// TIA Portal V17 export
// export: Created 2025-03-05T08:01:26.5756457Z, ExportSetting WithDefaults, DisplayName Totally Integrated Automation Portal, DisplayVersion V17 Update 8, DisplayName TIA Portal Openness, DisplayVersion V17 Update 8, DisplayName TIA Portal Version Control Interface, DisplayVersion V17, DisplayName SINAMICS Startdrive Advanced, DisplayVersion V17 SP2, DisplayName SINAMICS Startdrive G110M, G120, G120C, G120D, G120P, G115D, DisplayVersion V17 SP2, DisplayName SINAMICS Startdrive G130, G150, S120, S150, SINAMICS MV, S210, DisplayVersion V17 SP2, DisplayName STEP 7 Professional, DisplayVersion V17 Update 8, DisplayName SINUMERIK ONE STEP 7 Toolbox, DisplayVersion V17 Update 12, DisplayName SINUMERIK 840D sl STEP 7 Toolbox, DisplayVersion V17 Update 12, DisplayName STEP 7 Safety, DisplayVersion V17 Update 6, DisplayName WinCC Advanced, DisplayVersion V17 Update 8
FUNCTION "FC16015_METHOD_CALLS_U02_STA3_COAXIAL" : Void   // FC16015, LAD
{ S7_Optimized_Access := 'TRUE' }
VERSION : 0.1
// stored: AutoNumber false, IsIECCheckEnabled false, SetENOAutomatically false, UDAEnableTagReadback false
   VAR_TEMP
      AUX_WSTRING_PART_ID_STA3 : WString;
      AUX_WCHARS : Array[0..63] of WChar;
      index : Int;
      ALARM_AUX : Bool;
      TEMP_PULSE : Bool;
   END_VAR
   VAR_TEMP   // added for the SCL form of the ladder/FBD networks
      _w1 : Bool;
   END_VAR
BEGIN

REGION Network 1 (SCL): TRANSFORM TO WCHARS
   FOR #index := 0 TO 63 DO
       #AUX_WCHARS[#index] := CHAR_TO_WCHAR("DB8000_PART_STATUS".UNIT_02.STATION_3.PART_A.PART_ID[#index]);
   END_FOR;
END_REGION

REGION Network 2: TRANSFORM TO WSTRING
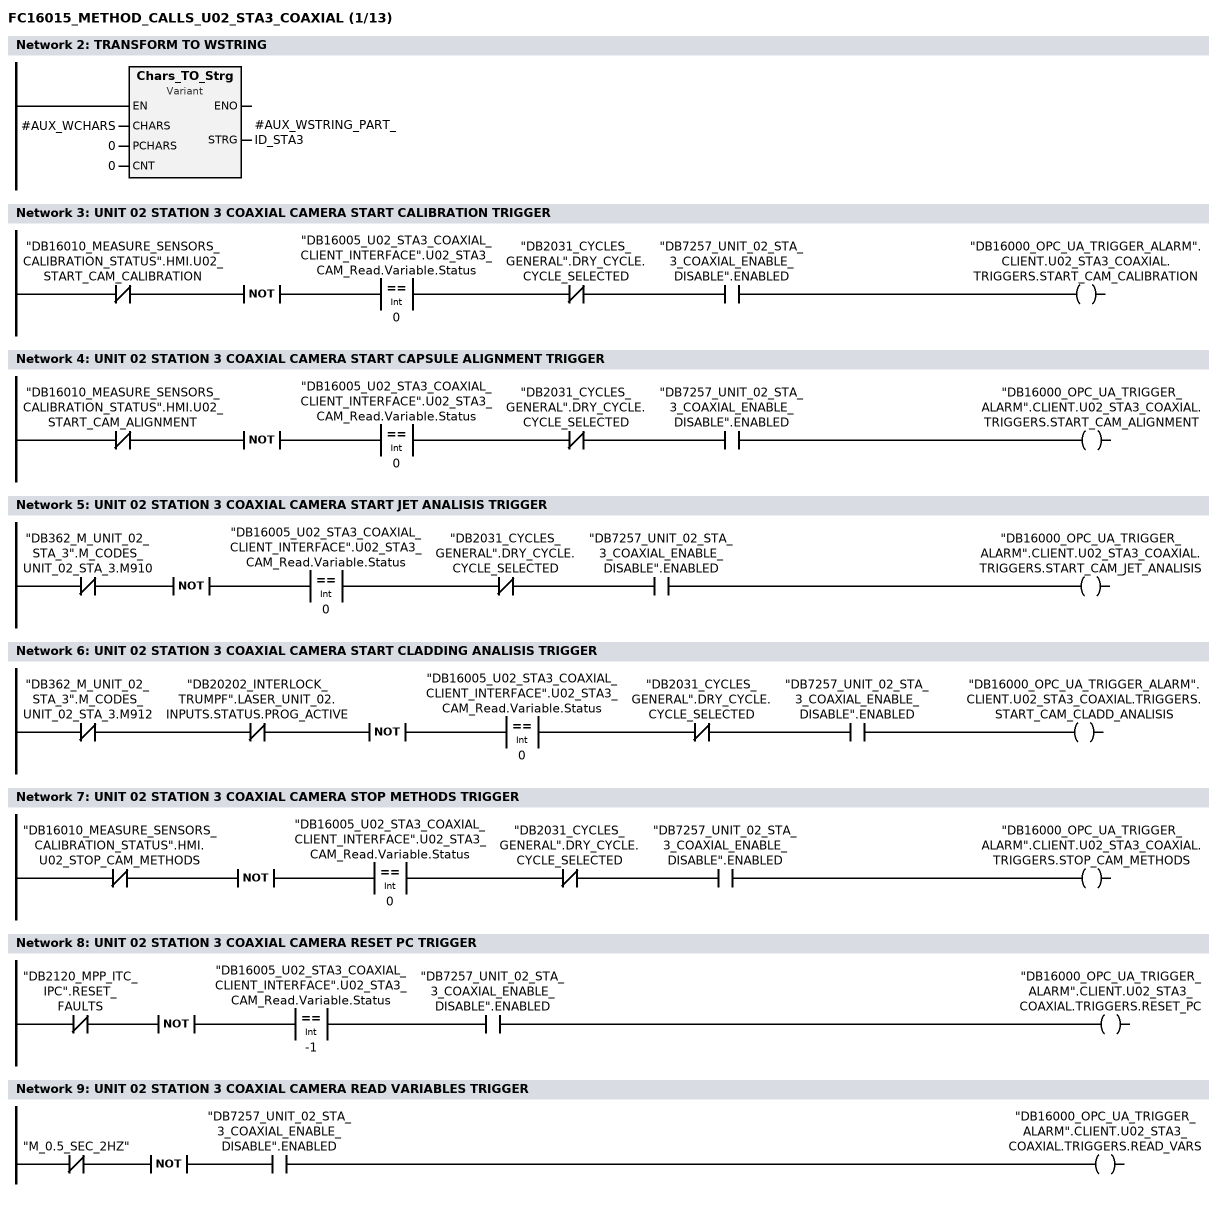
   RUNG wire#powerrail
      { S7_Templates := "[ptr_type := Variant, str_type := WString]" } Chars_TO_Strg(Chars := #AUX_WCHARS, pChars := 0, Cnt := 0, Strg => #AUX_WSTRING_PART_ID_STA3)
   END_RUNG
   // the same network as SCL:
   Chars_TO_Strg(Chars := #AUX_WCHARS, pChars := 0, Cnt := 0, Strg => #AUX_WSTRING_PART_ID_STA3);
END_REGION

REGION Network 3: UNIT 02 STATION 3 COAXIAL CAMERA START CALIBRATION TRIGGER
   RUNG wire#powerrail
      I_Contact( "DB16010_MEASURE_SENSORS_CALIBRATION_STATUS".HMI.U02_START_CAM_CALIBRATION )
      Not()
      { S7_Templates := "SrcType := Int" } EQ_Contact(in1 := "DB16005_U02_STA3_COAXIAL_CLIENT_INTERFACE".U02_STA3_CAM_Read.Variable.Status, in2 := 0)
      I_Contact( "DB2031_CYCLES_GENERAL".DRY_CYCLE.CYCLE_SELECTED )
      Contact( "DB7257_UNIT_02_STA_3_COAXIAL_ENABLE_DISABLE".ENABLED )
      Coil( "DB16000_OPC_UA_TRIGGER_ALARM".CLIENT.U02_STA3_COAXIAL.TRIGGERS.START_CAM_CALIBRATION )
   END_RUNG
   // the same network as SCL:
   "DB16000_OPC_UA_TRIGGER_ALARM".CLIENT.U02_STA3_COAXIAL.TRIGGERS.START_CAM_CALIBRATION := NOT (NOT "DB16010_MEASURE_SENSORS_CALIBRATION_STATUS".HMI.U02_START_CAM_CALIBRATION) AND ("DB16005_U02_STA3_COAXIAL_CLIENT_INTERFACE".U02_STA3_CAM_Read.Variable.Status = 0) AND NOT "DB2031_CYCLES_GENERAL".DRY_CYCLE.CYCLE_SELECTED AND "DB7257_UNIT_02_STA_3_COAXIAL_ENABLE_DISABLE".ENABLED;
END_REGION

REGION Network 4: UNIT 02 STATION 3 COAXIAL CAMERA START CAPSULE ALIGNMENT TRIGGER
   RUNG wire#powerrail
      I_Contact( "DB16010_MEASURE_SENSORS_CALIBRATION_STATUS".HMI.U02_START_CAM_ALIGNMENT )
      Not()
      { S7_Templates := "SrcType := Int" } EQ_Contact(in1 := "DB16005_U02_STA3_COAXIAL_CLIENT_INTERFACE".U02_STA3_CAM_Read.Variable.Status, in2 := 0)
      I_Contact( "DB2031_CYCLES_GENERAL".DRY_CYCLE.CYCLE_SELECTED )
      Contact( "DB7257_UNIT_02_STA_3_COAXIAL_ENABLE_DISABLE".ENABLED )
      Coil( "DB16000_OPC_UA_TRIGGER_ALARM".CLIENT.U02_STA3_COAXIAL.TRIGGERS.START_CAM_ALIGNMENT )
   END_RUNG
   // the same network as SCL:
   "DB16000_OPC_UA_TRIGGER_ALARM".CLIENT.U02_STA3_COAXIAL.TRIGGERS.START_CAM_ALIGNMENT := NOT (NOT "DB16010_MEASURE_SENSORS_CALIBRATION_STATUS".HMI.U02_START_CAM_ALIGNMENT) AND ("DB16005_U02_STA3_COAXIAL_CLIENT_INTERFACE".U02_STA3_CAM_Read.Variable.Status = 0) AND NOT "DB2031_CYCLES_GENERAL".DRY_CYCLE.CYCLE_SELECTED AND "DB7257_UNIT_02_STA_3_COAXIAL_ENABLE_DISABLE".ENABLED;
END_REGION

REGION Network 5: UNIT 02 STATION 3 COAXIAL CAMERA START JET ANALISIS TRIGGER
   RUNG wire#powerrail
      I_Contact( "DB362_M_UNIT_02_STA_3".M_CODES_UNIT_02_STA_3.M910 )
      Not()
      { S7_Templates := "SrcType := Int" } EQ_Contact(in1 := "DB16005_U02_STA3_COAXIAL_CLIENT_INTERFACE".U02_STA3_CAM_Read.Variable.Status, in2 := 0)
      I_Contact( "DB2031_CYCLES_GENERAL".DRY_CYCLE.CYCLE_SELECTED )
      Contact( "DB7257_UNIT_02_STA_3_COAXIAL_ENABLE_DISABLE".ENABLED )
      Coil( "DB16000_OPC_UA_TRIGGER_ALARM".CLIENT.U02_STA3_COAXIAL.TRIGGERS.START_CAM_JET_ANALISIS )
   END_RUNG
   // the same network as SCL:
   "DB16000_OPC_UA_TRIGGER_ALARM".CLIENT.U02_STA3_COAXIAL.TRIGGERS.START_CAM_JET_ANALISIS := NOT (NOT "DB362_M_UNIT_02_STA_3".M_CODES_UNIT_02_STA_3.M910) AND ("DB16005_U02_STA3_COAXIAL_CLIENT_INTERFACE".U02_STA3_CAM_Read.Variable.Status = 0) AND NOT "DB2031_CYCLES_GENERAL".DRY_CYCLE.CYCLE_SELECTED AND "DB7257_UNIT_02_STA_3_COAXIAL_ENABLE_DISABLE".ENABLED;
END_REGION

REGION Network 6: UNIT 02 STATION 3 COAXIAL CAMERA START CLADDING ANALISIS TRIGGER
   RUNG wire#powerrail
      I_Contact( "DB362_M_UNIT_02_STA_3".M_CODES_UNIT_02_STA_3.M912 )
      I_Contact( "DB20202_INTERLOCK_TRUMPF".LASER_UNIT_02.INPUTS.STATUS.PROG_ACTIVE )
      Not()
      { S7_Templates := "SrcType := Int" } EQ_Contact(in1 := "DB16005_U02_STA3_COAXIAL_CLIENT_INTERFACE".U02_STA3_CAM_Read.Variable.Status, in2 := 0)
      I_Contact( "DB2031_CYCLES_GENERAL".DRY_CYCLE.CYCLE_SELECTED )
      Contact( "DB7257_UNIT_02_STA_3_COAXIAL_ENABLE_DISABLE".ENABLED )
      Coil( "DB16000_OPC_UA_TRIGGER_ALARM".CLIENT.U02_STA3_COAXIAL.TRIGGERS.START_CAM_CLADD_ANALISIS )
   END_RUNG
   // the same network as SCL:
   "DB16000_OPC_UA_TRIGGER_ALARM".CLIENT.U02_STA3_COAXIAL.TRIGGERS.START_CAM_CLADD_ANALISIS := NOT (NOT "DB362_M_UNIT_02_STA_3".M_CODES_UNIT_02_STA_3.M912 AND NOT "DB20202_INTERLOCK_TRUMPF".LASER_UNIT_02.INPUTS.STATUS.PROG_ACTIVE) AND ("DB16005_U02_STA3_COAXIAL_CLIENT_INTERFACE".U02_STA3_CAM_Read.Variable.Status = 0) AND NOT "DB2031_CYCLES_GENERAL".DRY_CYCLE.CYCLE_SELECTED AND "DB7257_UNIT_02_STA_3_COAXIAL_ENABLE_DISABLE".ENABLED;
END_REGION

REGION Network 7: UNIT 02 STATION 3 COAXIAL CAMERA STOP METHODS TRIGGER
   RUNG wire#powerrail
      I_Contact( "DB16010_MEASURE_SENSORS_CALIBRATION_STATUS".HMI.U02_STOP_CAM_METHODS )
      Not()
      { S7_Templates := "SrcType := Int" } EQ_Contact(in1 := "DB16005_U02_STA3_COAXIAL_CLIENT_INTERFACE".U02_STA3_CAM_Read.Variable.Status, in2 := 0)
      I_Contact( "DB2031_CYCLES_GENERAL".DRY_CYCLE.CYCLE_SELECTED )
      Contact( "DB7257_UNIT_02_STA_3_COAXIAL_ENABLE_DISABLE".ENABLED )
      Coil( "DB16000_OPC_UA_TRIGGER_ALARM".CLIENT.U02_STA3_COAXIAL.TRIGGERS.STOP_CAM_METHODS )
   END_RUNG
   // the same network as SCL:
   "DB16000_OPC_UA_TRIGGER_ALARM".CLIENT.U02_STA3_COAXIAL.TRIGGERS.STOP_CAM_METHODS := NOT (NOT "DB16010_MEASURE_SENSORS_CALIBRATION_STATUS".HMI.U02_STOP_CAM_METHODS) AND ("DB16005_U02_STA3_COAXIAL_CLIENT_INTERFACE".U02_STA3_CAM_Read.Variable.Status = 0) AND NOT "DB2031_CYCLES_GENERAL".DRY_CYCLE.CYCLE_SELECTED AND "DB7257_UNIT_02_STA_3_COAXIAL_ENABLE_DISABLE".ENABLED;
END_REGION

REGION Network 8: UNIT 02 STATION 3 COAXIAL CAMERA RESET PC TRIGGER
   RUNG wire#powerrail
      I_Contact( "DB2120_MPP_ITC_IPC".RESET_FAULTS )
      Not()
      { S7_Templates := "SrcType := Int" } EQ_Contact(in1 := "DB16005_U02_STA3_COAXIAL_CLIENT_INTERFACE".U02_STA3_CAM_Read.Variable.Status, in2 := -1)
      Contact( "DB7257_UNIT_02_STA_3_COAXIAL_ENABLE_DISABLE".ENABLED )
      Coil( "DB16000_OPC_UA_TRIGGER_ALARM".CLIENT.U02_STA3_COAXIAL.TRIGGERS.RESET_PC )
   END_RUNG
   // the same network as SCL:
   "DB16000_OPC_UA_TRIGGER_ALARM".CLIENT.U02_STA3_COAXIAL.TRIGGERS.RESET_PC := NOT (NOT "DB2120_MPP_ITC_IPC".RESET_FAULTS) AND ("DB16005_U02_STA3_COAXIAL_CLIENT_INTERFACE".U02_STA3_CAM_Read.Variable.Status = (-1)) AND "DB7257_UNIT_02_STA_3_COAXIAL_ENABLE_DISABLE".ENABLED;
END_REGION

REGION Network 9: UNIT 02 STATION 3 COAXIAL CAMERA READ VARIABLES TRIGGER
   RUNG wire#powerrail
      I_Contact( "M_0.5_SEC_2HZ" )
      Not()
      Contact( "DB7257_UNIT_02_STA_3_COAXIAL_ENABLE_DISABLE".ENABLED )
      Coil( "DB16000_OPC_UA_TRIGGER_ALARM".CLIENT.U02_STA3_COAXIAL.TRIGGERS.READ_VARS )
   END_RUNG
   // the same network as SCL:
   "DB16000_OPC_UA_TRIGGER_ALARM".CLIENT.U02_STA3_COAXIAL.TRIGGERS.READ_VARS := NOT (NOT "M_0.5_SEC_2HZ") AND "DB7257_UNIT_02_STA_3_COAXIAL_ENABLE_DISABLE".ENABLED;
END_REGION

REGION Network 10: UNIT 02 STATION 3 COAXIAL CAMERA START CALIBRATION TRIGGER CALL-------------------------------------------------------
   // CAMBIAR POR EL METODO CORRECTO
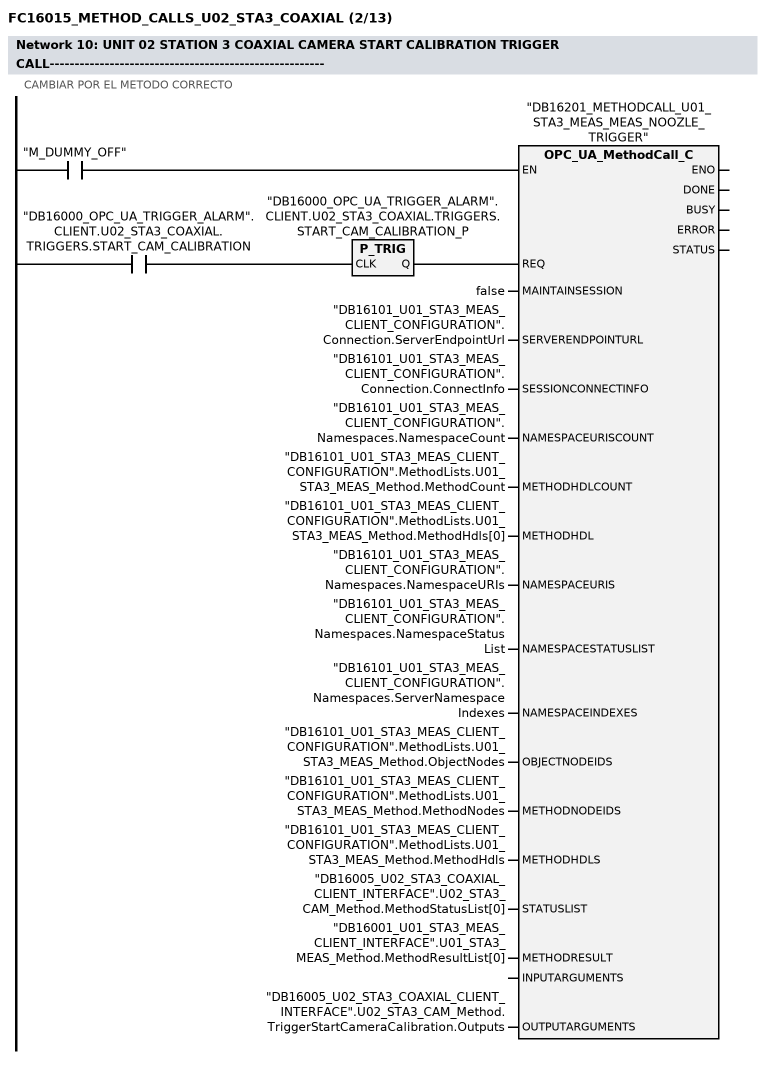
   RUNG wire#powerrail
      Contact( "M_DUMMY_OFF" )
      "DB16201_METHODCALL_U01_STA3_MEAS_MEAS_NOOZLE_TRIGGER".OPC_UA_MethodCall_C(REQ := wire#w1, MaintainSession := false, ServerEndpointUrl := "DB16101_U01_STA3_MEAS_CLIENT_CONFIGURATION".Connection.ServerEndpointUrl, SessionConnectInfo := "DB16101_U01_STA3_MEAS_CLIENT_CONFIGURATION".Connection.ConnectInfo, NamespaceUrisCount := "DB16101_U01_STA3_MEAS_CLIENT_CONFIGURATION".Namespaces.NamespaceCount, MethodHdlCount := "DB16101_U01_STA3_MEAS_CLIENT_CONFIGURATION".MethodLists.U01_STA3_MEAS_Method.MethodCount, MethodHdl := "DB16101_U01_STA3_MEAS_CLIENT_CONFIGURATION".MethodLists.U01_STA3_MEAS_Method.MethodHdls[0], NamespaceUris := "DB16101_U01_STA3_MEAS_CLIENT_CONFIGURATION".Namespaces.NamespaceURIs, NamespaceStatusList := "DB16101_U01_STA3_MEAS_CLIENT_CONFIGURATION".Namespaces.NamespaceStatusList, NamespaceIndexes := "DB16101_U01_STA3_MEAS_CLIENT_CONFIGURATION".Namespaces.ServerNamespaceIndexes, ObjectNodeIDs := "DB16101_U01_STA3_MEAS_CLIENT_CONFIGURATION".MethodLists.U01_STA3_MEAS_Method.ObjectNodes, MethodNodeIDs := "DB16101_U01_STA3_MEAS_CLIENT_CONFIGURATION".MethodLists.U01_STA3_MEAS_Method.MethodNodes, MethodHdls := "DB16101_U01_STA3_MEAS_CLIENT_CONFIGURATION".MethodLists.U01_STA3_MEAS_Method.MethodHdls, StatusList := "DB16005_U02_STA3_COAXIAL_CLIENT_INTERFACE".U02_STA3_CAM_Method.MethodStatusList[0], MethodResult := "DB16001_U01_STA3_MEAS_CLIENT_INTERFACE".U01_STA3_MEAS_Method.MethodResultList[0], InputArguments :=, OutputArguments := "DB16005_U02_STA3_COAXIAL_CLIENT_INTERFACE".U02_STA3_CAM_Method.TriggerStartCameraCalibration.Outputs, Done =>, Busy =>, Error =>, Status =>)
   END_RUNG
   RUNG wire#powerrail
      Contact( "DB16000_OPC_UA_TRIGGER_ALARM".CLIENT.U02_STA3_COAXIAL.TRIGGERS.START_CAM_CALIBRATION )
      P_Trig( "DB16000_OPC_UA_TRIGGER_ALARM".CLIENT.U02_STA3_COAXIAL.TRIGGERS.START_CAM_CALIBRATION_P )
   END_RUNG wire#w1
   // the same network as SCL:
   #_w1 := "DB16000_OPC_UA_TRIGGER_ALARM".CLIENT.U02_STA3_COAXIAL.TRIGGERS.START_CAM_CALIBRATION AND NOT "DB16000_OPC_UA_TRIGGER_ALARM".CLIENT.U02_STA3_COAXIAL.TRIGGERS.START_CAM_CALIBRATION_P;   // rising edge
   "DB16000_OPC_UA_TRIGGER_ALARM".CLIENT.U02_STA3_COAXIAL.TRIGGERS.START_CAM_CALIBRATION_P := "DB16000_OPC_UA_TRIGGER_ALARM".CLIENT.U02_STA3_COAXIAL.TRIGGERS.START_CAM_CALIBRATION;
   IF "M_DUMMY_OFF" THEN
       "DB16201_METHODCALL_U01_STA3_MEAS_MEAS_NOOZLE_TRIGGER"(REQ := #_w1,   // OPC_UA_MethodCall_C
                               MaintainSession := false,
                               ServerEndpointUrl := "DB16101_U01_STA3_MEAS_CLIENT_CONFIGURATION".Connection.ServerEndpointUrl,
                               SessionConnectInfo := "DB16101_U01_STA3_MEAS_CLIENT_CONFIGURATION".Connection.ConnectInfo,
                               NamespaceUrisCount := "DB16101_U01_STA3_MEAS_CLIENT_CONFIGURATION".Namespaces.NamespaceCount,
                               MethodHdlCount := "DB16101_U01_STA3_MEAS_CLIENT_CONFIGURATION".MethodLists.U01_STA3_MEAS_Method.MethodCount,
                               MethodHdl := "DB16101_U01_STA3_MEAS_CLIENT_CONFIGURATION".MethodLists.U01_STA3_MEAS_Method.MethodHdls[0],
                               NamespaceUris := "DB16101_U01_STA3_MEAS_CLIENT_CONFIGURATION".Namespaces.NamespaceURIs,
                               NamespaceStatusList := "DB16101_U01_STA3_MEAS_CLIENT_CONFIGURATION".Namespaces.NamespaceStatusList,
                               NamespaceIndexes := "DB16101_U01_STA3_MEAS_CLIENT_CONFIGURATION".Namespaces.ServerNamespaceIndexes,
                               ObjectNodeIDs := "DB16101_U01_STA3_MEAS_CLIENT_CONFIGURATION".MethodLists.U01_STA3_MEAS_Method.ObjectNodes,
                               MethodNodeIDs := "DB16101_U01_STA3_MEAS_CLIENT_CONFIGURATION".MethodLists.U01_STA3_MEAS_Method.MethodNodes,
                               MethodHdls := "DB16101_U01_STA3_MEAS_CLIENT_CONFIGURATION".MethodLists.U01_STA3_MEAS_Method.MethodHdls,
                               StatusList := "DB16005_U02_STA3_COAXIAL_CLIENT_INTERFACE".U02_STA3_CAM_Method.MethodStatusList[0],
                               MethodResult := "DB16001_U01_STA3_MEAS_CLIENT_INTERFACE".U01_STA3_MEAS_Method.MethodResultList[0],
                               OutputArguments := "DB16005_U02_STA3_COAXIAL_CLIENT_INTERFACE".U02_STA3_CAM_Method.TriggerStartCameraCalibration.Outputs);
   END_IF;
END_REGION

REGION Network 11: UNIT 02 STATION 3 COAXIAL CAMERA START CAPSULE ALIGNMENT TRIGGER CALL----------------------------------------
   // CAMBIAR POR EL METODO CORRECTO
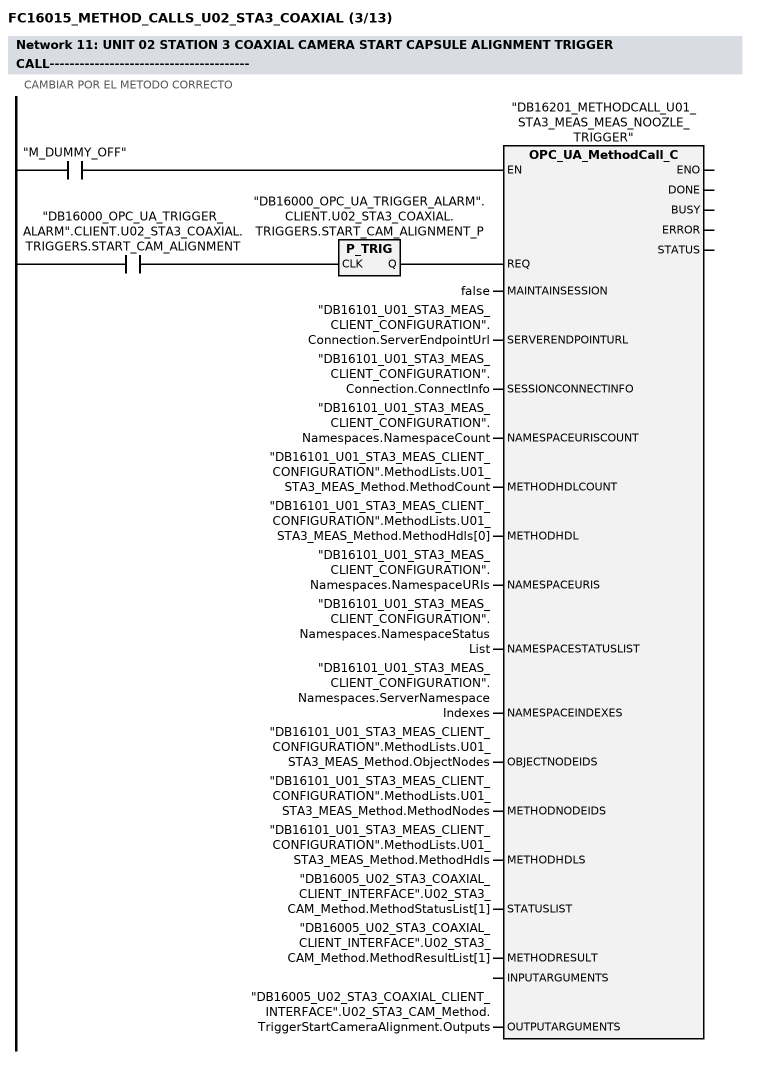
   RUNG wire#powerrail
      Contact( "M_DUMMY_OFF" )
      "DB16201_METHODCALL_U01_STA3_MEAS_MEAS_NOOZLE_TRIGGER".OPC_UA_MethodCall_C(REQ := wire#w1, MaintainSession := false, ServerEndpointUrl := "DB16101_U01_STA3_MEAS_CLIENT_CONFIGURATION".Connection.ServerEndpointUrl, SessionConnectInfo := "DB16101_U01_STA3_MEAS_CLIENT_CONFIGURATION".Connection.ConnectInfo, NamespaceUrisCount := "DB16101_U01_STA3_MEAS_CLIENT_CONFIGURATION".Namespaces.NamespaceCount, MethodHdlCount := "DB16101_U01_STA3_MEAS_CLIENT_CONFIGURATION".MethodLists.U01_STA3_MEAS_Method.MethodCount, MethodHdl := "DB16101_U01_STA3_MEAS_CLIENT_CONFIGURATION".MethodLists.U01_STA3_MEAS_Method.MethodHdls[0], NamespaceUris := "DB16101_U01_STA3_MEAS_CLIENT_CONFIGURATION".Namespaces.NamespaceURIs, NamespaceStatusList := "DB16101_U01_STA3_MEAS_CLIENT_CONFIGURATION".Namespaces.NamespaceStatusList, NamespaceIndexes := "DB16101_U01_STA3_MEAS_CLIENT_CONFIGURATION".Namespaces.ServerNamespaceIndexes, ObjectNodeIDs := "DB16101_U01_STA3_MEAS_CLIENT_CONFIGURATION".MethodLists.U01_STA3_MEAS_Method.ObjectNodes, MethodNodeIDs := "DB16101_U01_STA3_MEAS_CLIENT_CONFIGURATION".MethodLists.U01_STA3_MEAS_Method.MethodNodes, MethodHdls := "DB16101_U01_STA3_MEAS_CLIENT_CONFIGURATION".MethodLists.U01_STA3_MEAS_Method.MethodHdls, StatusList := "DB16005_U02_STA3_COAXIAL_CLIENT_INTERFACE".U02_STA3_CAM_Method.MethodStatusList[1], MethodResult := "DB16005_U02_STA3_COAXIAL_CLIENT_INTERFACE".U02_STA3_CAM_Method.MethodResultList[1], InputArguments :=, OutputArguments := "DB16005_U02_STA3_COAXIAL_CLIENT_INTERFACE".U02_STA3_CAM_Method.TriggerStartCameraAlignment.Outputs, Done =>, Busy =>, Error =>, Status =>)
   END_RUNG
   RUNG wire#powerrail
      Contact( "DB16000_OPC_UA_TRIGGER_ALARM".CLIENT.U02_STA3_COAXIAL.TRIGGERS.START_CAM_ALIGNMENT )
      P_Trig( "DB16000_OPC_UA_TRIGGER_ALARM".CLIENT.U02_STA3_COAXIAL.TRIGGERS.START_CAM_ALIGNMENT_P )
   END_RUNG wire#w1
   // the same network as SCL:
   #_w1 := "DB16000_OPC_UA_TRIGGER_ALARM".CLIENT.U02_STA3_COAXIAL.TRIGGERS.START_CAM_ALIGNMENT AND NOT "DB16000_OPC_UA_TRIGGER_ALARM".CLIENT.U02_STA3_COAXIAL.TRIGGERS.START_CAM_ALIGNMENT_P;   // rising edge
   "DB16000_OPC_UA_TRIGGER_ALARM".CLIENT.U02_STA3_COAXIAL.TRIGGERS.START_CAM_ALIGNMENT_P := "DB16000_OPC_UA_TRIGGER_ALARM".CLIENT.U02_STA3_COAXIAL.TRIGGERS.START_CAM_ALIGNMENT;
   IF "M_DUMMY_OFF" THEN
       "DB16201_METHODCALL_U01_STA3_MEAS_MEAS_NOOZLE_TRIGGER"(REQ := #_w1,   // OPC_UA_MethodCall_C
                               MaintainSession := false,
                               ServerEndpointUrl := "DB16101_U01_STA3_MEAS_CLIENT_CONFIGURATION".Connection.ServerEndpointUrl,
                               SessionConnectInfo := "DB16101_U01_STA3_MEAS_CLIENT_CONFIGURATION".Connection.ConnectInfo,
                               NamespaceUrisCount := "DB16101_U01_STA3_MEAS_CLIENT_CONFIGURATION".Namespaces.NamespaceCount,
                               MethodHdlCount := "DB16101_U01_STA3_MEAS_CLIENT_CONFIGURATION".MethodLists.U01_STA3_MEAS_Method.MethodCount,
                               MethodHdl := "DB16101_U01_STA3_MEAS_CLIENT_CONFIGURATION".MethodLists.U01_STA3_MEAS_Method.MethodHdls[0],
                               NamespaceUris := "DB16101_U01_STA3_MEAS_CLIENT_CONFIGURATION".Namespaces.NamespaceURIs,
                               NamespaceStatusList := "DB16101_U01_STA3_MEAS_CLIENT_CONFIGURATION".Namespaces.NamespaceStatusList,
                               NamespaceIndexes := "DB16101_U01_STA3_MEAS_CLIENT_CONFIGURATION".Namespaces.ServerNamespaceIndexes,
                               ObjectNodeIDs := "DB16101_U01_STA3_MEAS_CLIENT_CONFIGURATION".MethodLists.U01_STA3_MEAS_Method.ObjectNodes,
                               MethodNodeIDs := "DB16101_U01_STA3_MEAS_CLIENT_CONFIGURATION".MethodLists.U01_STA3_MEAS_Method.MethodNodes,
                               MethodHdls := "DB16101_U01_STA3_MEAS_CLIENT_CONFIGURATION".MethodLists.U01_STA3_MEAS_Method.MethodHdls,
                               StatusList := "DB16005_U02_STA3_COAXIAL_CLIENT_INTERFACE".U02_STA3_CAM_Method.MethodStatusList[1],
                               MethodResult := "DB16005_U02_STA3_COAXIAL_CLIENT_INTERFACE".U02_STA3_CAM_Method.MethodResultList[1],
                               OutputArguments := "DB16005_U02_STA3_COAXIAL_CLIENT_INTERFACE".U02_STA3_CAM_Method.TriggerStartCameraAlignment.Outputs);
   END_IF;
END_REGION

REGION Network 12: UNIT 02 STATION 3 COAXIAL CAMERA START JET ANALISIS TRIGGER CALL-------------------------------------------------------
   // CAMBIAR POR EL METODO CORRECTO
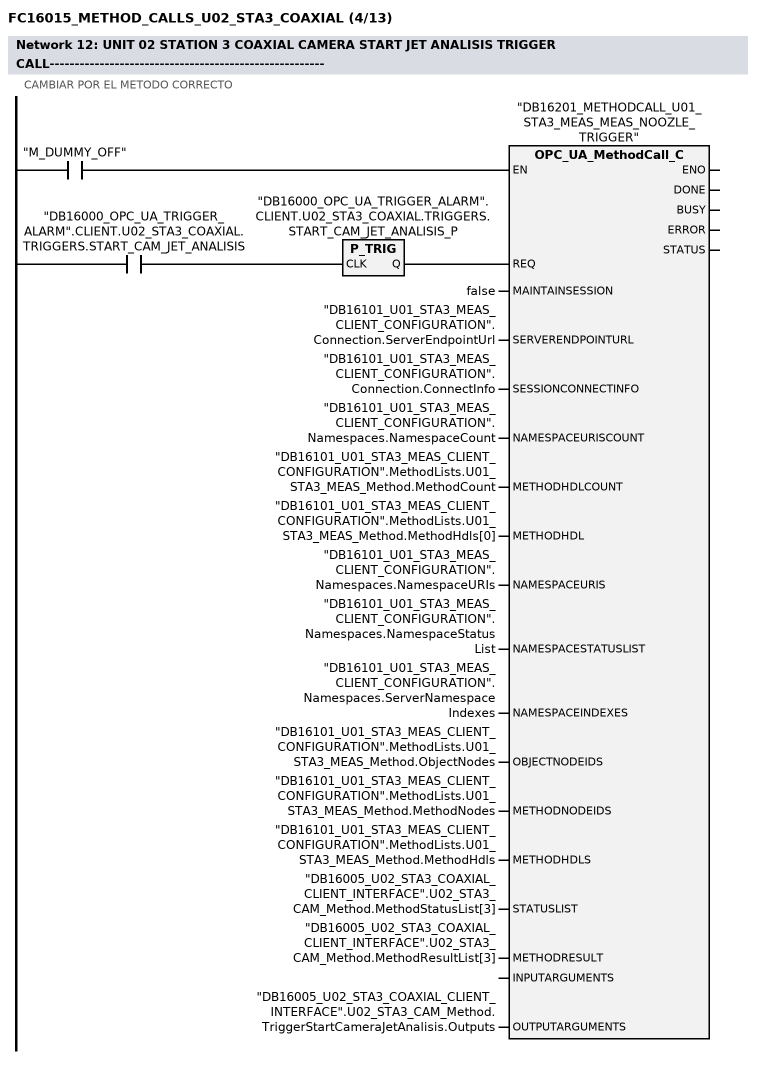
   RUNG wire#powerrail
      Contact( "M_DUMMY_OFF" )
      "DB16201_METHODCALL_U01_STA3_MEAS_MEAS_NOOZLE_TRIGGER".OPC_UA_MethodCall_C(REQ := wire#w1, MaintainSession := false, ServerEndpointUrl := "DB16101_U01_STA3_MEAS_CLIENT_CONFIGURATION".Connection.ServerEndpointUrl, SessionConnectInfo := "DB16101_U01_STA3_MEAS_CLIENT_CONFIGURATION".Connection.ConnectInfo, NamespaceUrisCount := "DB16101_U01_STA3_MEAS_CLIENT_CONFIGURATION".Namespaces.NamespaceCount, MethodHdlCount := "DB16101_U01_STA3_MEAS_CLIENT_CONFIGURATION".MethodLists.U01_STA3_MEAS_Method.MethodCount, MethodHdl := "DB16101_U01_STA3_MEAS_CLIENT_CONFIGURATION".MethodLists.U01_STA3_MEAS_Method.MethodHdls[0], NamespaceUris := "DB16101_U01_STA3_MEAS_CLIENT_CONFIGURATION".Namespaces.NamespaceURIs, NamespaceStatusList := "DB16101_U01_STA3_MEAS_CLIENT_CONFIGURATION".Namespaces.NamespaceStatusList, NamespaceIndexes := "DB16101_U01_STA3_MEAS_CLIENT_CONFIGURATION".Namespaces.ServerNamespaceIndexes, ObjectNodeIDs := "DB16101_U01_STA3_MEAS_CLIENT_CONFIGURATION".MethodLists.U01_STA3_MEAS_Method.ObjectNodes, MethodNodeIDs := "DB16101_U01_STA3_MEAS_CLIENT_CONFIGURATION".MethodLists.U01_STA3_MEAS_Method.MethodNodes, MethodHdls := "DB16101_U01_STA3_MEAS_CLIENT_CONFIGURATION".MethodLists.U01_STA3_MEAS_Method.MethodHdls, StatusList := "DB16005_U02_STA3_COAXIAL_CLIENT_INTERFACE".U02_STA3_CAM_Method.MethodStatusList[3], MethodResult := "DB16005_U02_STA3_COAXIAL_CLIENT_INTERFACE".U02_STA3_CAM_Method.MethodResultList[3], InputArguments :=, OutputArguments := "DB16005_U02_STA3_COAXIAL_CLIENT_INTERFACE".U02_STA3_CAM_Method.TriggerStartCameraJetAnalisis.Outputs, Done =>, Busy =>, Error =>, Status =>)
   END_RUNG
   RUNG wire#powerrail
      Contact( "DB16000_OPC_UA_TRIGGER_ALARM".CLIENT.U02_STA3_COAXIAL.TRIGGERS.START_CAM_JET_ANALISIS )
      P_Trig( "DB16000_OPC_UA_TRIGGER_ALARM".CLIENT.U02_STA3_COAXIAL.TRIGGERS.START_CAM_JET_ANALISIS_P )
   END_RUNG wire#w1
   // the same network as SCL:
   #_w1 := "DB16000_OPC_UA_TRIGGER_ALARM".CLIENT.U02_STA3_COAXIAL.TRIGGERS.START_CAM_JET_ANALISIS AND NOT "DB16000_OPC_UA_TRIGGER_ALARM".CLIENT.U02_STA3_COAXIAL.TRIGGERS.START_CAM_JET_ANALISIS_P;   // rising edge
   "DB16000_OPC_UA_TRIGGER_ALARM".CLIENT.U02_STA3_COAXIAL.TRIGGERS.START_CAM_JET_ANALISIS_P := "DB16000_OPC_UA_TRIGGER_ALARM".CLIENT.U02_STA3_COAXIAL.TRIGGERS.START_CAM_JET_ANALISIS;
   IF "M_DUMMY_OFF" THEN
       "DB16201_METHODCALL_U01_STA3_MEAS_MEAS_NOOZLE_TRIGGER"(REQ := #_w1,   // OPC_UA_MethodCall_C
                               MaintainSession := false,
                               ServerEndpointUrl := "DB16101_U01_STA3_MEAS_CLIENT_CONFIGURATION".Connection.ServerEndpointUrl,
                               SessionConnectInfo := "DB16101_U01_STA3_MEAS_CLIENT_CONFIGURATION".Connection.ConnectInfo,
                               NamespaceUrisCount := "DB16101_U01_STA3_MEAS_CLIENT_CONFIGURATION".Namespaces.NamespaceCount,
                               MethodHdlCount := "DB16101_U01_STA3_MEAS_CLIENT_CONFIGURATION".MethodLists.U01_STA3_MEAS_Method.MethodCount,
                               MethodHdl := "DB16101_U01_STA3_MEAS_CLIENT_CONFIGURATION".MethodLists.U01_STA3_MEAS_Method.MethodHdls[0],
                               NamespaceUris := "DB16101_U01_STA3_MEAS_CLIENT_CONFIGURATION".Namespaces.NamespaceURIs,
                               NamespaceStatusList := "DB16101_U01_STA3_MEAS_CLIENT_CONFIGURATION".Namespaces.NamespaceStatusList,
                               NamespaceIndexes := "DB16101_U01_STA3_MEAS_CLIENT_CONFIGURATION".Namespaces.ServerNamespaceIndexes,
                               ObjectNodeIDs := "DB16101_U01_STA3_MEAS_CLIENT_CONFIGURATION".MethodLists.U01_STA3_MEAS_Method.ObjectNodes,
                               MethodNodeIDs := "DB16101_U01_STA3_MEAS_CLIENT_CONFIGURATION".MethodLists.U01_STA3_MEAS_Method.MethodNodes,
                               MethodHdls := "DB16101_U01_STA3_MEAS_CLIENT_CONFIGURATION".MethodLists.U01_STA3_MEAS_Method.MethodHdls,
                               StatusList := "DB16005_U02_STA3_COAXIAL_CLIENT_INTERFACE".U02_STA3_CAM_Method.MethodStatusList[3],
                               MethodResult := "DB16005_U02_STA3_COAXIAL_CLIENT_INTERFACE".U02_STA3_CAM_Method.MethodResultList[3],
                               OutputArguments := "DB16005_U02_STA3_COAXIAL_CLIENT_INTERFACE".U02_STA3_CAM_Method.TriggerStartCameraJetAnalisis.Outputs);
   END_IF;
END_REGION

REGION Network 13: UNIT 02 STATION 3 COAXIAL CAMERA START CLADDING ANALISIS TRIGGER CALL------------------------------------------
   // CAMBIAR POR EL METODO CORRECTO
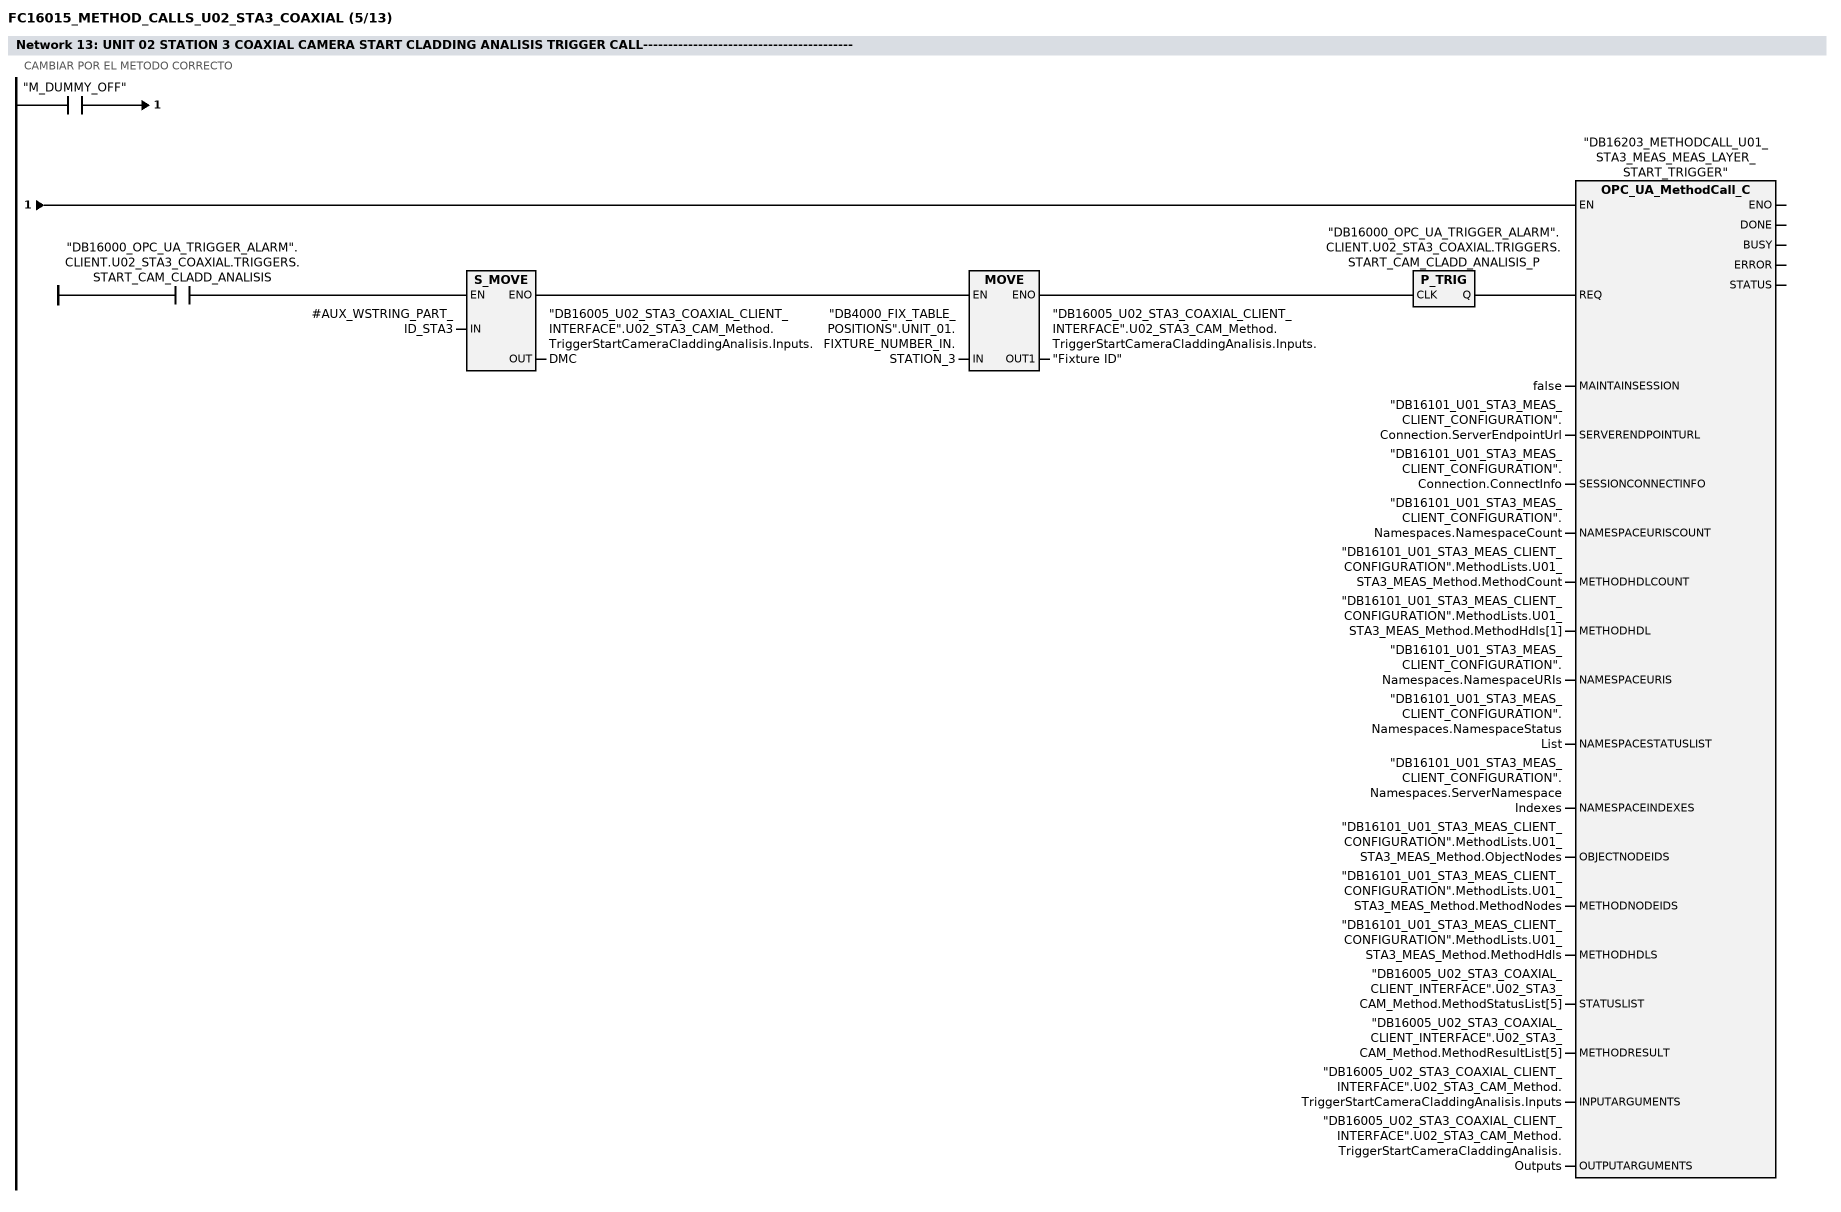
   RUNG wire#powerrail
      Contact( "M_DUMMY_OFF" )
      "DB16203_METHODCALL_U01_STA3_MEAS_MEAS_LAYER_START_TRIGGER".OPC_UA_MethodCall_C(REQ := wire#w1, MaintainSession := false, ServerEndpointUrl := "DB16101_U01_STA3_MEAS_CLIENT_CONFIGURATION".Connection.ServerEndpointUrl, SessionConnectInfo := "DB16101_U01_STA3_MEAS_CLIENT_CONFIGURATION".Connection.ConnectInfo, NamespaceUrisCount := "DB16101_U01_STA3_MEAS_CLIENT_CONFIGURATION".Namespaces.NamespaceCount, MethodHdlCount := "DB16101_U01_STA3_MEAS_CLIENT_CONFIGURATION".MethodLists.U01_STA3_MEAS_Method.MethodCount, MethodHdl := "DB16101_U01_STA3_MEAS_CLIENT_CONFIGURATION".MethodLists.U01_STA3_MEAS_Method.MethodHdls[1], NamespaceUris := "DB16101_U01_STA3_MEAS_CLIENT_CONFIGURATION".Namespaces.NamespaceURIs, NamespaceStatusList := "DB16101_U01_STA3_MEAS_CLIENT_CONFIGURATION".Namespaces.NamespaceStatusList, NamespaceIndexes := "DB16101_U01_STA3_MEAS_CLIENT_CONFIGURATION".Namespaces.ServerNamespaceIndexes, ObjectNodeIDs := "DB16101_U01_STA3_MEAS_CLIENT_CONFIGURATION".MethodLists.U01_STA3_MEAS_Method.ObjectNodes, MethodNodeIDs := "DB16101_U01_STA3_MEAS_CLIENT_CONFIGURATION".MethodLists.U01_STA3_MEAS_Method.MethodNodes, MethodHdls := "DB16101_U01_STA3_MEAS_CLIENT_CONFIGURATION".MethodLists.U01_STA3_MEAS_Method.MethodHdls, StatusList := "DB16005_U02_STA3_COAXIAL_CLIENT_INTERFACE".U02_STA3_CAM_Method.MethodStatusList[5], MethodResult := "DB16005_U02_STA3_COAXIAL_CLIENT_INTERFACE".U02_STA3_CAM_Method.MethodResultList[5], InputArguments := "DB16005_U02_STA3_COAXIAL_CLIENT_INTERFACE".U02_STA3_CAM_Method.TriggerStartCameraCladdingAnalisis.Inputs, OutputArguments := "DB16005_U02_STA3_COAXIAL_CLIENT_INTERFACE".U02_STA3_CAM_Method.TriggerStartCameraCladdingAnalisis.Outputs, Done =>, Busy =>, Error =>, Status =>)
   END_RUNG
   RUNG wire#powerrail
      Contact( "DB16000_OPC_UA_TRIGGER_ALARM".CLIENT.U02_STA3_COAXIAL.TRIGGERS.START_CAM_CLADD_ANALISIS )
      S_Move(in := #AUX_WSTRING_PART_ID_STA3, out => "DB16005_U02_STA3_COAXIAL_CLIENT_INTERFACE".U02_STA3_CAM_Method.TriggerStartCameraCladdingAnalisis.Inputs.DMC)
      Move(in := "DB4000_FIX_TABLE_POSITIONS".UNIT_01.FIXTURE_NUMBER_IN.STATION_3, out1 => "DB16005_U02_STA3_COAXIAL_CLIENT_INTERFACE".U02_STA3_CAM_Method.TriggerStartCameraCladdingAnalisis.Inputs."Fixture ID")
      P_Trig( "DB16000_OPC_UA_TRIGGER_ALARM".CLIENT.U02_STA3_COAXIAL.TRIGGERS.START_CAM_CLADD_ANALISIS_P )
   END_RUNG wire#w1
   // the same network as SCL:
   IF "DB16000_OPC_UA_TRIGGER_ALARM".CLIENT.U02_STA3_COAXIAL.TRIGGERS.START_CAM_CLADD_ANALISIS THEN
       "DB16005_U02_STA3_COAXIAL_CLIENT_INTERFACE".U02_STA3_CAM_Method.TriggerStartCameraCladdingAnalisis.Inputs.DMC := #AUX_WSTRING_PART_ID_STA3;
       "DB16005_U02_STA3_COAXIAL_CLIENT_INTERFACE".U02_STA3_CAM_Method.TriggerStartCameraCladdingAnalisis.Inputs."Fixture ID" := "DB4000_FIX_TABLE_POSITIONS".UNIT_01.FIXTURE_NUMBER_IN.STATION_3;
   END_IF;
   #_w1 := "DB16000_OPC_UA_TRIGGER_ALARM".CLIENT.U02_STA3_COAXIAL.TRIGGERS.START_CAM_CLADD_ANALISIS AND NOT "DB16000_OPC_UA_TRIGGER_ALARM".CLIENT.U02_STA3_COAXIAL.TRIGGERS.START_CAM_CLADD_ANALISIS_P;   // rising edge
   "DB16000_OPC_UA_TRIGGER_ALARM".CLIENT.U02_STA3_COAXIAL.TRIGGERS.START_CAM_CLADD_ANALISIS_P := "DB16000_OPC_UA_TRIGGER_ALARM".CLIENT.U02_STA3_COAXIAL.TRIGGERS.START_CAM_CLADD_ANALISIS;
   IF "M_DUMMY_OFF" THEN
       "DB16203_METHODCALL_U01_STA3_MEAS_MEAS_LAYER_START_TRIGGER"(REQ := #_w1,   // OPC_UA_MethodCall_C
                               MaintainSession := false,
                               ServerEndpointUrl := "DB16101_U01_STA3_MEAS_CLIENT_CONFIGURATION".Connection.ServerEndpointUrl,
                               SessionConnectInfo := "DB16101_U01_STA3_MEAS_CLIENT_CONFIGURATION".Connection.ConnectInfo,
                               NamespaceUrisCount := "DB16101_U01_STA3_MEAS_CLIENT_CONFIGURATION".Namespaces.NamespaceCount,
                               MethodHdlCount := "DB16101_U01_STA3_MEAS_CLIENT_CONFIGURATION".MethodLists.U01_STA3_MEAS_Method.MethodCount,
                               MethodHdl := "DB16101_U01_STA3_MEAS_CLIENT_CONFIGURATION".MethodLists.U01_STA3_MEAS_Method.MethodHdls[1],
                               NamespaceUris := "DB16101_U01_STA3_MEAS_CLIENT_CONFIGURATION".Namespaces.NamespaceURIs,
                               NamespaceStatusList := "DB16101_U01_STA3_MEAS_CLIENT_CONFIGURATION".Namespaces.NamespaceStatusList,
                               NamespaceIndexes := "DB16101_U01_STA3_MEAS_CLIENT_CONFIGURATION".Namespaces.ServerNamespaceIndexes,
                               ObjectNodeIDs := "DB16101_U01_STA3_MEAS_CLIENT_CONFIGURATION".MethodLists.U01_STA3_MEAS_Method.ObjectNodes,
                               MethodNodeIDs := "DB16101_U01_STA3_MEAS_CLIENT_CONFIGURATION".MethodLists.U01_STA3_MEAS_Method.MethodNodes,
                               MethodHdls := "DB16101_U01_STA3_MEAS_CLIENT_CONFIGURATION".MethodLists.U01_STA3_MEAS_Method.MethodHdls,
                               StatusList := "DB16005_U02_STA3_COAXIAL_CLIENT_INTERFACE".U02_STA3_CAM_Method.MethodStatusList[5],
                               MethodResult := "DB16005_U02_STA3_COAXIAL_CLIENT_INTERFACE".U02_STA3_CAM_Method.MethodResultList[5],
                               InputArguments := "DB16005_U02_STA3_COAXIAL_CLIENT_INTERFACE".U02_STA3_CAM_Method.TriggerStartCameraCladdingAnalisis.Inputs,
                               OutputArguments := "DB16005_U02_STA3_COAXIAL_CLIENT_INTERFACE".U02_STA3_CAM_Method.TriggerStartCameraCladdingAnalisis.Outputs);
   END_IF;
END_REGION

REGION Network 14: UNIT 02 STATION 3 COAXIAL CAMERA STOP METHODS TRIGGER CALL-------------------------------------------------
   // CAMBIAR POR EL METODO CORRECTO
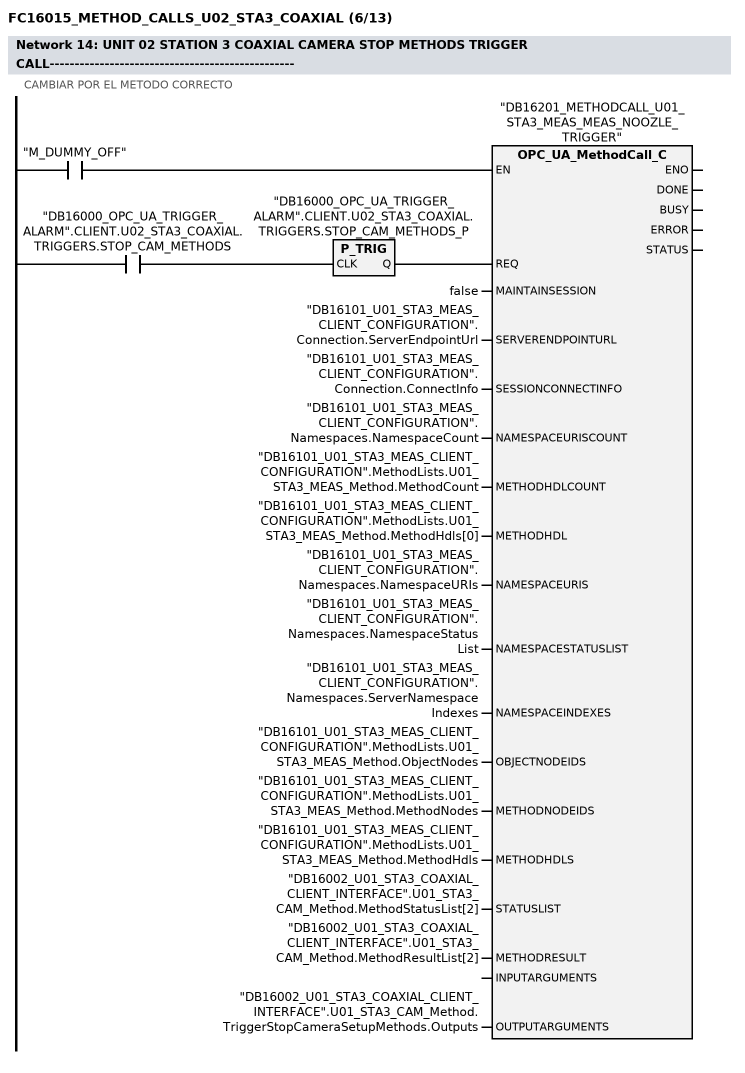
   RUNG wire#powerrail
      Contact( "M_DUMMY_OFF" )
      "DB16201_METHODCALL_U01_STA3_MEAS_MEAS_NOOZLE_TRIGGER".OPC_UA_MethodCall_C(REQ := wire#w1, MaintainSession := false, ServerEndpointUrl := "DB16101_U01_STA3_MEAS_CLIENT_CONFIGURATION".Connection.ServerEndpointUrl, SessionConnectInfo := "DB16101_U01_STA3_MEAS_CLIENT_CONFIGURATION".Connection.ConnectInfo, NamespaceUrisCount := "DB16101_U01_STA3_MEAS_CLIENT_CONFIGURATION".Namespaces.NamespaceCount, MethodHdlCount := "DB16101_U01_STA3_MEAS_CLIENT_CONFIGURATION".MethodLists.U01_STA3_MEAS_Method.MethodCount, MethodHdl := "DB16101_U01_STA3_MEAS_CLIENT_CONFIGURATION".MethodLists.U01_STA3_MEAS_Method.MethodHdls[0], NamespaceUris := "DB16101_U01_STA3_MEAS_CLIENT_CONFIGURATION".Namespaces.NamespaceURIs, NamespaceStatusList := "DB16101_U01_STA3_MEAS_CLIENT_CONFIGURATION".Namespaces.NamespaceStatusList, NamespaceIndexes := "DB16101_U01_STA3_MEAS_CLIENT_CONFIGURATION".Namespaces.ServerNamespaceIndexes, ObjectNodeIDs := "DB16101_U01_STA3_MEAS_CLIENT_CONFIGURATION".MethodLists.U01_STA3_MEAS_Method.ObjectNodes, MethodNodeIDs := "DB16101_U01_STA3_MEAS_CLIENT_CONFIGURATION".MethodLists.U01_STA3_MEAS_Method.MethodNodes, MethodHdls := "DB16101_U01_STA3_MEAS_CLIENT_CONFIGURATION".MethodLists.U01_STA3_MEAS_Method.MethodHdls, StatusList := "DB16002_U01_STA3_COAXIAL_CLIENT_INTERFACE".U01_STA3_CAM_Method.MethodStatusList[2], MethodResult := "DB16002_U01_STA3_COAXIAL_CLIENT_INTERFACE".U01_STA3_CAM_Method.MethodResultList[2], InputArguments :=, OutputArguments := "DB16002_U01_STA3_COAXIAL_CLIENT_INTERFACE".U01_STA3_CAM_Method.TriggerStopCameraSetupMethods.Outputs, Done =>, Busy =>, Error =>, Status =>)
   END_RUNG
   RUNG wire#powerrail
      Contact( "DB16000_OPC_UA_TRIGGER_ALARM".CLIENT.U02_STA3_COAXIAL.TRIGGERS.STOP_CAM_METHODS )
      P_Trig( "DB16000_OPC_UA_TRIGGER_ALARM".CLIENT.U02_STA3_COAXIAL.TRIGGERS.STOP_CAM_METHODS_P )
   END_RUNG wire#w1
   // the same network as SCL:
   #_w1 := "DB16000_OPC_UA_TRIGGER_ALARM".CLIENT.U02_STA3_COAXIAL.TRIGGERS.STOP_CAM_METHODS AND NOT "DB16000_OPC_UA_TRIGGER_ALARM".CLIENT.U02_STA3_COAXIAL.TRIGGERS.STOP_CAM_METHODS_P;   // rising edge
   "DB16000_OPC_UA_TRIGGER_ALARM".CLIENT.U02_STA3_COAXIAL.TRIGGERS.STOP_CAM_METHODS_P := "DB16000_OPC_UA_TRIGGER_ALARM".CLIENT.U02_STA3_COAXIAL.TRIGGERS.STOP_CAM_METHODS;
   IF "M_DUMMY_OFF" THEN
       "DB16201_METHODCALL_U01_STA3_MEAS_MEAS_NOOZLE_TRIGGER"(REQ := #_w1,   // OPC_UA_MethodCall_C
                               MaintainSession := false,
                               ServerEndpointUrl := "DB16101_U01_STA3_MEAS_CLIENT_CONFIGURATION".Connection.ServerEndpointUrl,
                               SessionConnectInfo := "DB16101_U01_STA3_MEAS_CLIENT_CONFIGURATION".Connection.ConnectInfo,
                               NamespaceUrisCount := "DB16101_U01_STA3_MEAS_CLIENT_CONFIGURATION".Namespaces.NamespaceCount,
                               MethodHdlCount := "DB16101_U01_STA3_MEAS_CLIENT_CONFIGURATION".MethodLists.U01_STA3_MEAS_Method.MethodCount,
                               MethodHdl := "DB16101_U01_STA3_MEAS_CLIENT_CONFIGURATION".MethodLists.U01_STA3_MEAS_Method.MethodHdls[0],
                               NamespaceUris := "DB16101_U01_STA3_MEAS_CLIENT_CONFIGURATION".Namespaces.NamespaceURIs,
                               NamespaceStatusList := "DB16101_U01_STA3_MEAS_CLIENT_CONFIGURATION".Namespaces.NamespaceStatusList,
                               NamespaceIndexes := "DB16101_U01_STA3_MEAS_CLIENT_CONFIGURATION".Namespaces.ServerNamespaceIndexes,
                               ObjectNodeIDs := "DB16101_U01_STA3_MEAS_CLIENT_CONFIGURATION".MethodLists.U01_STA3_MEAS_Method.ObjectNodes,
                               MethodNodeIDs := "DB16101_U01_STA3_MEAS_CLIENT_CONFIGURATION".MethodLists.U01_STA3_MEAS_Method.MethodNodes,
                               MethodHdls := "DB16101_U01_STA3_MEAS_CLIENT_CONFIGURATION".MethodLists.U01_STA3_MEAS_Method.MethodHdls,
                               StatusList := "DB16002_U01_STA3_COAXIAL_CLIENT_INTERFACE".U01_STA3_CAM_Method.MethodStatusList[2],
                               MethodResult := "DB16002_U01_STA3_COAXIAL_CLIENT_INTERFACE".U01_STA3_CAM_Method.MethodResultList[2],
                               OutputArguments := "DB16002_U01_STA3_COAXIAL_CLIENT_INTERFACE".U01_STA3_CAM_Method.TriggerStopCameraSetupMethods.Outputs);
   END_IF;
END_REGION

REGION Network 15: UNIT 02 STATION 3 COAXIAL CAMERA RESET PC TRIGGER CALL------------------------------------------------------------------------
   // CAMBIAR POR EL METODO CORRECTO
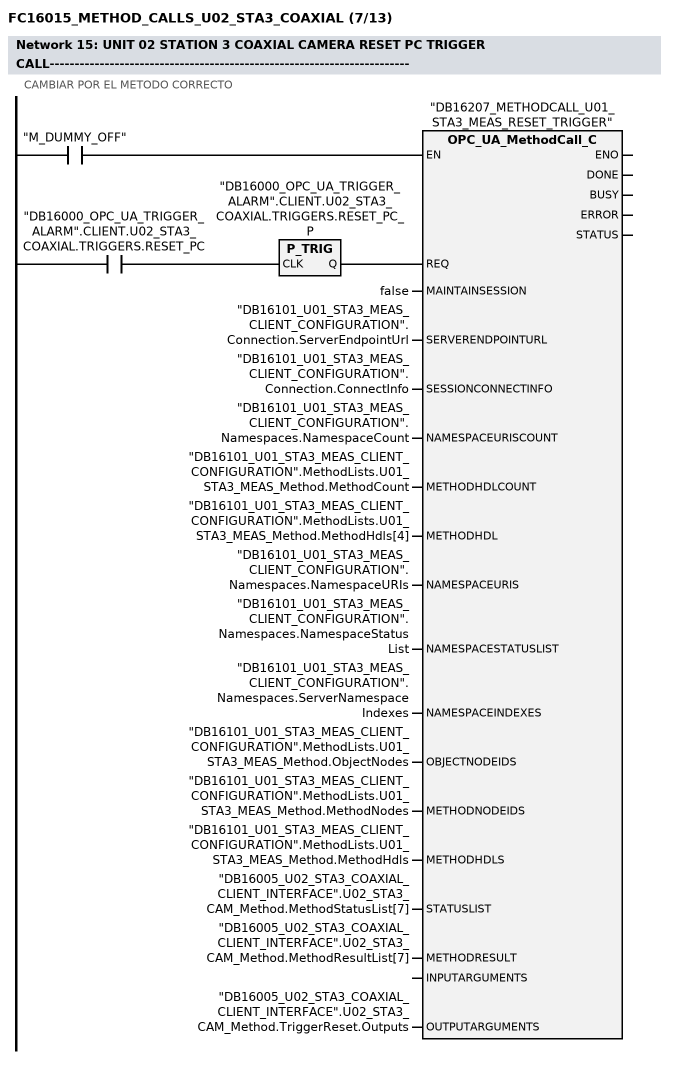
   RUNG wire#powerrail
      Contact( "M_DUMMY_OFF" )
      "DB16207_METHODCALL_U01_STA3_MEAS_RESET_TRIGGER".OPC_UA_MethodCall_C(REQ := wire#w1, MaintainSession := false, ServerEndpointUrl := "DB16101_U01_STA3_MEAS_CLIENT_CONFIGURATION".Connection.ServerEndpointUrl, SessionConnectInfo := "DB16101_U01_STA3_MEAS_CLIENT_CONFIGURATION".Connection.ConnectInfo, NamespaceUrisCount := "DB16101_U01_STA3_MEAS_CLIENT_CONFIGURATION".Namespaces.NamespaceCount, MethodHdlCount := "DB16101_U01_STA3_MEAS_CLIENT_CONFIGURATION".MethodLists.U01_STA3_MEAS_Method.MethodCount, MethodHdl := "DB16101_U01_STA3_MEAS_CLIENT_CONFIGURATION".MethodLists.U01_STA3_MEAS_Method.MethodHdls[4], NamespaceUris := "DB16101_U01_STA3_MEAS_CLIENT_CONFIGURATION".Namespaces.NamespaceURIs, NamespaceStatusList := "DB16101_U01_STA3_MEAS_CLIENT_CONFIGURATION".Namespaces.NamespaceStatusList, NamespaceIndexes := "DB16101_U01_STA3_MEAS_CLIENT_CONFIGURATION".Namespaces.ServerNamespaceIndexes, ObjectNodeIDs := "DB16101_U01_STA3_MEAS_CLIENT_CONFIGURATION".MethodLists.U01_STA3_MEAS_Method.ObjectNodes, MethodNodeIDs := "DB16101_U01_STA3_MEAS_CLIENT_CONFIGURATION".MethodLists.U01_STA3_MEAS_Method.MethodNodes, MethodHdls := "DB16101_U01_STA3_MEAS_CLIENT_CONFIGURATION".MethodLists.U01_STA3_MEAS_Method.MethodHdls, StatusList := "DB16005_U02_STA3_COAXIAL_CLIENT_INTERFACE".U02_STA3_CAM_Method.MethodStatusList[7], MethodResult := "DB16005_U02_STA3_COAXIAL_CLIENT_INTERFACE".U02_STA3_CAM_Method.MethodResultList[7], InputArguments :=, OutputArguments := "DB16005_U02_STA3_COAXIAL_CLIENT_INTERFACE".U02_STA3_CAM_Method.TriggerReset.Outputs, Done =>, Busy =>, Error =>, Status =>)
   END_RUNG
   RUNG wire#powerrail
      Contact( "DB16000_OPC_UA_TRIGGER_ALARM".CLIENT.U02_STA3_COAXIAL.TRIGGERS.RESET_PC )
      P_Trig( "DB16000_OPC_UA_TRIGGER_ALARM".CLIENT.U02_STA3_COAXIAL.TRIGGERS.RESET_PC_P )
   END_RUNG wire#w1
   // the same network as SCL:
   #_w1 := "DB16000_OPC_UA_TRIGGER_ALARM".CLIENT.U02_STA3_COAXIAL.TRIGGERS.RESET_PC AND NOT "DB16000_OPC_UA_TRIGGER_ALARM".CLIENT.U02_STA3_COAXIAL.TRIGGERS.RESET_PC_P;   // rising edge
   "DB16000_OPC_UA_TRIGGER_ALARM".CLIENT.U02_STA3_COAXIAL.TRIGGERS.RESET_PC_P := "DB16000_OPC_UA_TRIGGER_ALARM".CLIENT.U02_STA3_COAXIAL.TRIGGERS.RESET_PC;
   IF "M_DUMMY_OFF" THEN
       "DB16207_METHODCALL_U01_STA3_MEAS_RESET_TRIGGER"(REQ := #_w1,   // OPC_UA_MethodCall_C
                               MaintainSession := false,
                               ServerEndpointUrl := "DB16101_U01_STA3_MEAS_CLIENT_CONFIGURATION".Connection.ServerEndpointUrl,
                               SessionConnectInfo := "DB16101_U01_STA3_MEAS_CLIENT_CONFIGURATION".Connection.ConnectInfo,
                               NamespaceUrisCount := "DB16101_U01_STA3_MEAS_CLIENT_CONFIGURATION".Namespaces.NamespaceCount,
                               MethodHdlCount := "DB16101_U01_STA3_MEAS_CLIENT_CONFIGURATION".MethodLists.U01_STA3_MEAS_Method.MethodCount,
                               MethodHdl := "DB16101_U01_STA3_MEAS_CLIENT_CONFIGURATION".MethodLists.U01_STA3_MEAS_Method.MethodHdls[4],
                               NamespaceUris := "DB16101_U01_STA3_MEAS_CLIENT_CONFIGURATION".Namespaces.NamespaceURIs,
                               NamespaceStatusList := "DB16101_U01_STA3_MEAS_CLIENT_CONFIGURATION".Namespaces.NamespaceStatusList,
                               NamespaceIndexes := "DB16101_U01_STA3_MEAS_CLIENT_CONFIGURATION".Namespaces.ServerNamespaceIndexes,
                               ObjectNodeIDs := "DB16101_U01_STA3_MEAS_CLIENT_CONFIGURATION".MethodLists.U01_STA3_MEAS_Method.ObjectNodes,
                               MethodNodeIDs := "DB16101_U01_STA3_MEAS_CLIENT_CONFIGURATION".MethodLists.U01_STA3_MEAS_Method.MethodNodes,
                               MethodHdls := "DB16101_U01_STA3_MEAS_CLIENT_CONFIGURATION".MethodLists.U01_STA3_MEAS_Method.MethodHdls,
                               StatusList := "DB16005_U02_STA3_COAXIAL_CLIENT_INTERFACE".U02_STA3_CAM_Method.MethodStatusList[7],
                               MethodResult := "DB16005_U02_STA3_COAXIAL_CLIENT_INTERFACE".U02_STA3_CAM_Method.MethodResultList[7],
                               OutputArguments := "DB16005_U02_STA3_COAXIAL_CLIENT_INTERFACE".U02_STA3_CAM_Method.TriggerReset.Outputs);
   END_IF;
END_REGION

REGION Network 16: UNIT 02 STATION 3 COAXIAL CAMERA READ VARIABLES TRIGGER CALL----------------------------------------------------------
   // CAMBIAR POR EL METODO CORRECTO
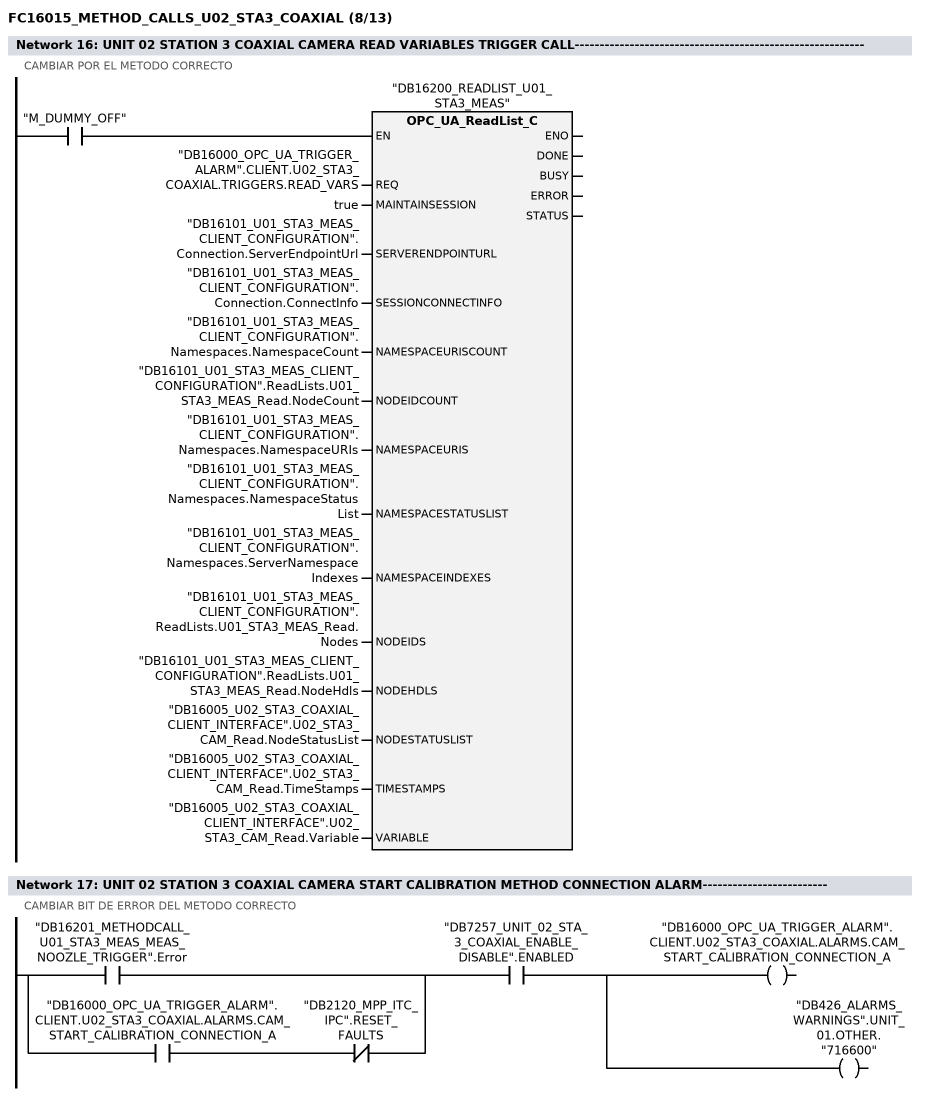
   RUNG wire#powerrail
      Contact( "M_DUMMY_OFF" )
      "DB16200_READLIST_U01_STA3_MEAS".OPC_UA_ReadList_C(REQ := "DB16000_OPC_UA_TRIGGER_ALARM".CLIENT.U02_STA3_COAXIAL.TRIGGERS.READ_VARS, MaintainSession := true, ServerEndpointUrl := "DB16101_U01_STA3_MEAS_CLIENT_CONFIGURATION".Connection.ServerEndpointUrl, SessionConnectInfo := "DB16101_U01_STA3_MEAS_CLIENT_CONFIGURATION".Connection.ConnectInfo, NamespaceUrisCount := "DB16101_U01_STA3_MEAS_CLIENT_CONFIGURATION".Namespaces.NamespaceCount, NodeIDCount := "DB16101_U01_STA3_MEAS_CLIENT_CONFIGURATION".ReadLists.U01_STA3_MEAS_Read.NodeCount, NamespaceUris := "DB16101_U01_STA3_MEAS_CLIENT_CONFIGURATION".Namespaces.NamespaceURIs, NamespaceStatusList := "DB16101_U01_STA3_MEAS_CLIENT_CONFIGURATION".Namespaces.NamespaceStatusList, NamespaceIndexes := "DB16101_U01_STA3_MEAS_CLIENT_CONFIGURATION".Namespaces.ServerNamespaceIndexes, NodeIDs := "DB16101_U01_STA3_MEAS_CLIENT_CONFIGURATION".ReadLists.U01_STA3_MEAS_Read.Nodes, NodeHdls := "DB16101_U01_STA3_MEAS_CLIENT_CONFIGURATION".ReadLists.U01_STA3_MEAS_Read.NodeHdls, NodeStatusList := "DB16005_U02_STA3_COAXIAL_CLIENT_INTERFACE".U02_STA3_CAM_Read.NodeStatusList, Timestamps := "DB16005_U02_STA3_COAXIAL_CLIENT_INTERFACE".U02_STA3_CAM_Read.TimeStamps, Variable := "DB16005_U02_STA3_COAXIAL_CLIENT_INTERFACE".U02_STA3_CAM_Read.Variable, Done =>, Busy =>, Error =>, Status =>)
   END_RUNG
   // the same network as SCL:
   IF "M_DUMMY_OFF" THEN
       "DB16200_READLIST_U01_STA3_MEAS"(REQ := "DB16000_OPC_UA_TRIGGER_ALARM".CLIENT.U02_STA3_COAXIAL.TRIGGERS.READ_VARS,   // OPC_UA_ReadList_C
                               MaintainSession := true,
                               ServerEndpointUrl := "DB16101_U01_STA3_MEAS_CLIENT_CONFIGURATION".Connection.ServerEndpointUrl,
                               SessionConnectInfo := "DB16101_U01_STA3_MEAS_CLIENT_CONFIGURATION".Connection.ConnectInfo,
                               NamespaceUrisCount := "DB16101_U01_STA3_MEAS_CLIENT_CONFIGURATION".Namespaces.NamespaceCount,
                               NodeIDCount := "DB16101_U01_STA3_MEAS_CLIENT_CONFIGURATION".ReadLists.U01_STA3_MEAS_Read.NodeCount,
                               NamespaceUris := "DB16101_U01_STA3_MEAS_CLIENT_CONFIGURATION".Namespaces.NamespaceURIs,
                               NamespaceStatusList := "DB16101_U01_STA3_MEAS_CLIENT_CONFIGURATION".Namespaces.NamespaceStatusList,
                               NamespaceIndexes := "DB16101_U01_STA3_MEAS_CLIENT_CONFIGURATION".Namespaces.ServerNamespaceIndexes,
                               NodeIDs := "DB16101_U01_STA3_MEAS_CLIENT_CONFIGURATION".ReadLists.U01_STA3_MEAS_Read.Nodes,
                               NodeHdls := "DB16101_U01_STA3_MEAS_CLIENT_CONFIGURATION".ReadLists.U01_STA3_MEAS_Read.NodeHdls,
                               NodeStatusList := "DB16005_U02_STA3_COAXIAL_CLIENT_INTERFACE".U02_STA3_CAM_Read.NodeStatusList,
                               Timestamps := "DB16005_U02_STA3_COAXIAL_CLIENT_INTERFACE".U02_STA3_CAM_Read.TimeStamps,
                               Variable := "DB16005_U02_STA3_COAXIAL_CLIENT_INTERFACE".U02_STA3_CAM_Read.Variable);
   END_IF;
END_REGION

REGION Network 17: UNIT 02 STATION 3 COAXIAL CAMERA START CALIBRATION METHOD CONNECTION ALARM-------------------------
   // CAMBIAR BIT DE ERROR DEL METODO CORRECTO
   RUNG wire#powerrail
      Contact( "DB16201_METHODCALL_U01_STA3_MEAS_MEAS_NOOZLE_TRIGGER".Error )
      wire#w1
      Contact( "DB7257_UNIT_02_STA_3_COAXIAL_ENABLE_DISABLE".ENABLED )
      wire#w2
      Coil( "DB16000_OPC_UA_TRIGGER_ALARM".CLIENT.U02_STA3_COAXIAL.ALARMS.CAM_START_CALIBRATION_CONNECTION_A )
   END_RUNG
   RUNG wire#powerrail
      Contact( "DB16000_OPC_UA_TRIGGER_ALARM".CLIENT.U02_STA3_COAXIAL.ALARMS.CAM_START_CALIBRATION_CONNECTION_A )
      I_Contact( "DB2120_MPP_ITC_IPC".RESET_FAULTS )
   END_RUNG wire#w1
   RUNG wire#w2
      Coil( "DB426_ALARMS_WARNINGS".UNIT_01.OTHER."716600" )
   END_RUNG
   // the same network as SCL:
   "DB16000_OPC_UA_TRIGGER_ALARM".CLIENT.U02_STA3_COAXIAL.ALARMS.CAM_START_CALIBRATION_CONNECTION_A := ("DB16201_METHODCALL_U01_STA3_MEAS_MEAS_NOOZLE_TRIGGER".Error OR ("DB16000_OPC_UA_TRIGGER_ALARM".CLIENT.U02_STA3_COAXIAL.ALARMS.CAM_START_CALIBRATION_CONNECTION_A AND NOT "DB2120_MPP_ITC_IPC".RESET_FAULTS)) AND "DB7257_UNIT_02_STA_3_COAXIAL_ENABLE_DISABLE".ENABLED;
   "DB426_ALARMS_WARNINGS".UNIT_01.OTHER."716600" := "DB16000_OPC_UA_TRIGGER_ALARM".CLIENT.U02_STA3_COAXIAL.ALARMS.CAM_START_CALIBRATION_CONNECTION_A;
END_REGION

REGION Network 18: UNIT 02 STATION 3 COAXIAL CAMERA START CALIBRATION METHOD WORKING OR BLOCKED ALARM--------
   // CAMBIAR BIT DE DONE DEL METODO CORRECTO
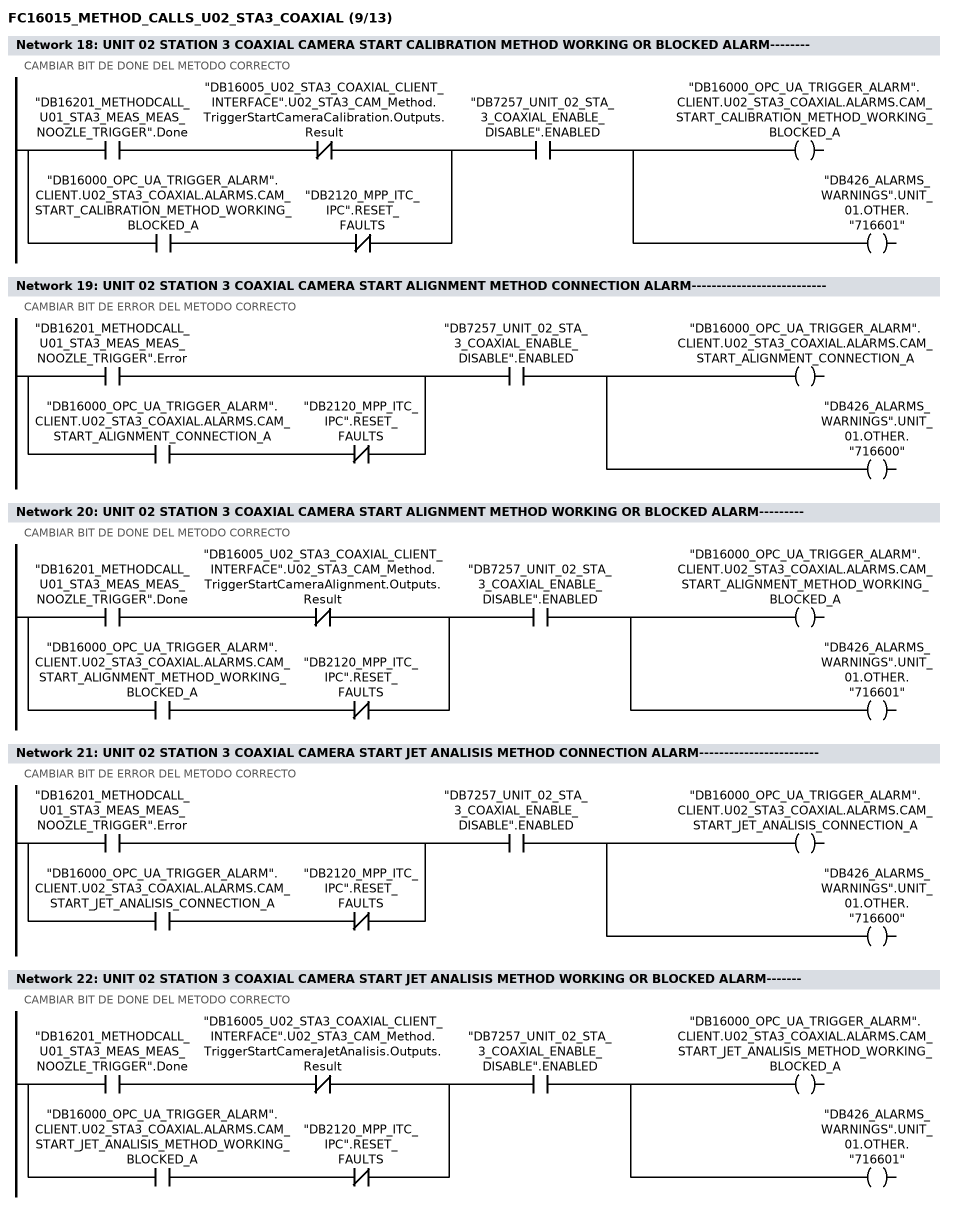
   RUNG wire#powerrail
      Contact( "DB16201_METHODCALL_U01_STA3_MEAS_MEAS_NOOZLE_TRIGGER".Done )
      I_Contact( "DB16005_U02_STA3_COAXIAL_CLIENT_INTERFACE".U02_STA3_CAM_Method.TriggerStartCameraCalibration.Outputs.Result )
      wire#w1
      Contact( "DB7257_UNIT_02_STA_3_COAXIAL_ENABLE_DISABLE".ENABLED )
      wire#w2
      Coil( "DB16000_OPC_UA_TRIGGER_ALARM".CLIENT.U02_STA3_COAXIAL.ALARMS.CAM_START_CALIBRATION_METHOD_WORKING_BLOCKED_A )
   END_RUNG
   RUNG wire#powerrail
      Contact( "DB16000_OPC_UA_TRIGGER_ALARM".CLIENT.U02_STA3_COAXIAL.ALARMS.CAM_START_CALIBRATION_METHOD_WORKING_BLOCKED_A )
      I_Contact( "DB2120_MPP_ITC_IPC".RESET_FAULTS )
   END_RUNG wire#w1
   RUNG wire#w2
      Coil( "DB426_ALARMS_WARNINGS".UNIT_01.OTHER."716601" )
   END_RUNG
   // the same network as SCL:
   "DB16000_OPC_UA_TRIGGER_ALARM".CLIENT.U02_STA3_COAXIAL.ALARMS.CAM_START_CALIBRATION_METHOD_WORKING_BLOCKED_A := (("DB16201_METHODCALL_U01_STA3_MEAS_MEAS_NOOZLE_TRIGGER".Done AND NOT "DB16005_U02_STA3_COAXIAL_CLIENT_INTERFACE".U02_STA3_CAM_Method.TriggerStartCameraCalibration.Outputs.Result) OR ("DB16000_OPC_UA_TRIGGER_ALARM".CLIENT.U02_STA3_COAXIAL.ALARMS.CAM_START_CALIBRATION_METHOD_WORKING_BLOCKED_A AND NOT "DB2120_MPP_ITC_IPC".RESET_FAULTS)) AND "DB7257_UNIT_02_STA_3_COAXIAL_ENABLE_DISABLE".ENABLED;
   "DB426_ALARMS_WARNINGS".UNIT_01.OTHER."716601" := "DB16000_OPC_UA_TRIGGER_ALARM".CLIENT.U02_STA3_COAXIAL.ALARMS.CAM_START_CALIBRATION_METHOD_WORKING_BLOCKED_A;
END_REGION

REGION Network 19: UNIT 02 STATION 3 COAXIAL CAMERA START ALIGNMENT METHOD CONNECTION ALARM---------------------------
   // CAMBIAR BIT DE ERROR DEL METODO CORRECTO
   RUNG wire#powerrail
      Contact( "DB16201_METHODCALL_U01_STA3_MEAS_MEAS_NOOZLE_TRIGGER".Error )
      wire#w1
      Contact( "DB7257_UNIT_02_STA_3_COAXIAL_ENABLE_DISABLE".ENABLED )
      wire#w2
      Coil( "DB16000_OPC_UA_TRIGGER_ALARM".CLIENT.U02_STA3_COAXIAL.ALARMS.CAM_START_ALIGNMENT_CONNECTION_A )
   END_RUNG
   RUNG wire#powerrail
      Contact( "DB16000_OPC_UA_TRIGGER_ALARM".CLIENT.U02_STA3_COAXIAL.ALARMS.CAM_START_ALIGNMENT_CONNECTION_A )
      I_Contact( "DB2120_MPP_ITC_IPC".RESET_FAULTS )
   END_RUNG wire#w1
   RUNG wire#w2
      Coil( "DB426_ALARMS_WARNINGS".UNIT_01.OTHER."716600" )
   END_RUNG
   // the same network as SCL:
   "DB16000_OPC_UA_TRIGGER_ALARM".CLIENT.U02_STA3_COAXIAL.ALARMS.CAM_START_ALIGNMENT_CONNECTION_A := ("DB16201_METHODCALL_U01_STA3_MEAS_MEAS_NOOZLE_TRIGGER".Error OR ("DB16000_OPC_UA_TRIGGER_ALARM".CLIENT.U02_STA3_COAXIAL.ALARMS.CAM_START_ALIGNMENT_CONNECTION_A AND NOT "DB2120_MPP_ITC_IPC".RESET_FAULTS)) AND "DB7257_UNIT_02_STA_3_COAXIAL_ENABLE_DISABLE".ENABLED;
   "DB426_ALARMS_WARNINGS".UNIT_01.OTHER."716600" := "DB16000_OPC_UA_TRIGGER_ALARM".CLIENT.U02_STA3_COAXIAL.ALARMS.CAM_START_ALIGNMENT_CONNECTION_A;
END_REGION

REGION Network 20: UNIT 02 STATION 3 COAXIAL CAMERA START ALIGNMENT METHOD WORKING OR BLOCKED ALARM---------
   // CAMBIAR BIT DE DONE DEL METODO CORRECTO
   RUNG wire#powerrail
      Contact( "DB16201_METHODCALL_U01_STA3_MEAS_MEAS_NOOZLE_TRIGGER".Done )
      I_Contact( "DB16005_U02_STA3_COAXIAL_CLIENT_INTERFACE".U02_STA3_CAM_Method.TriggerStartCameraAlignment.Outputs.Result )
      wire#w1
      Contact( "DB7257_UNIT_02_STA_3_COAXIAL_ENABLE_DISABLE".ENABLED )
      wire#w2
      Coil( "DB16000_OPC_UA_TRIGGER_ALARM".CLIENT.U02_STA3_COAXIAL.ALARMS.CAM_START_ALIGNMENT_METHOD_WORKING_BLOCKED_A )
   END_RUNG
   RUNG wire#powerrail
      Contact( "DB16000_OPC_UA_TRIGGER_ALARM".CLIENT.U02_STA3_COAXIAL.ALARMS.CAM_START_ALIGNMENT_METHOD_WORKING_BLOCKED_A )
      I_Contact( "DB2120_MPP_ITC_IPC".RESET_FAULTS )
   END_RUNG wire#w1
   RUNG wire#w2
      Coil( "DB426_ALARMS_WARNINGS".UNIT_01.OTHER."716601" )
   END_RUNG
   // the same network as SCL:
   "DB16000_OPC_UA_TRIGGER_ALARM".CLIENT.U02_STA3_COAXIAL.ALARMS.CAM_START_ALIGNMENT_METHOD_WORKING_BLOCKED_A := (("DB16201_METHODCALL_U01_STA3_MEAS_MEAS_NOOZLE_TRIGGER".Done AND NOT "DB16005_U02_STA3_COAXIAL_CLIENT_INTERFACE".U02_STA3_CAM_Method.TriggerStartCameraAlignment.Outputs.Result) OR ("DB16000_OPC_UA_TRIGGER_ALARM".CLIENT.U02_STA3_COAXIAL.ALARMS.CAM_START_ALIGNMENT_METHOD_WORKING_BLOCKED_A AND NOT "DB2120_MPP_ITC_IPC".RESET_FAULTS)) AND "DB7257_UNIT_02_STA_3_COAXIAL_ENABLE_DISABLE".ENABLED;
   "DB426_ALARMS_WARNINGS".UNIT_01.OTHER."716601" := "DB16000_OPC_UA_TRIGGER_ALARM".CLIENT.U02_STA3_COAXIAL.ALARMS.CAM_START_ALIGNMENT_METHOD_WORKING_BLOCKED_A;
END_REGION

REGION Network 21: UNIT 02 STATION 3 COAXIAL CAMERA START JET ANALISIS METHOD CONNECTION ALARM------------------------
   // CAMBIAR BIT DE ERROR DEL METODO CORRECTO
   RUNG wire#powerrail
      Contact( "DB16201_METHODCALL_U01_STA3_MEAS_MEAS_NOOZLE_TRIGGER".Error )
      wire#w1
      Contact( "DB7257_UNIT_02_STA_3_COAXIAL_ENABLE_DISABLE".ENABLED )
      wire#w2
      Coil( "DB16000_OPC_UA_TRIGGER_ALARM".CLIENT.U02_STA3_COAXIAL.ALARMS.CAM_START_JET_ANALISIS_CONNECTION_A )
   END_RUNG
   RUNG wire#powerrail
      Contact( "DB16000_OPC_UA_TRIGGER_ALARM".CLIENT.U02_STA3_COAXIAL.ALARMS.CAM_START_JET_ANALISIS_CONNECTION_A )
      I_Contact( "DB2120_MPP_ITC_IPC".RESET_FAULTS )
   END_RUNG wire#w1
   RUNG wire#w2
      Coil( "DB426_ALARMS_WARNINGS".UNIT_01.OTHER."716600" )
   END_RUNG
   // the same network as SCL:
   "DB16000_OPC_UA_TRIGGER_ALARM".CLIENT.U02_STA3_COAXIAL.ALARMS.CAM_START_JET_ANALISIS_CONNECTION_A := ("DB16201_METHODCALL_U01_STA3_MEAS_MEAS_NOOZLE_TRIGGER".Error OR ("DB16000_OPC_UA_TRIGGER_ALARM".CLIENT.U02_STA3_COAXIAL.ALARMS.CAM_START_JET_ANALISIS_CONNECTION_A AND NOT "DB2120_MPP_ITC_IPC".RESET_FAULTS)) AND "DB7257_UNIT_02_STA_3_COAXIAL_ENABLE_DISABLE".ENABLED;
   "DB426_ALARMS_WARNINGS".UNIT_01.OTHER."716600" := "DB16000_OPC_UA_TRIGGER_ALARM".CLIENT.U02_STA3_COAXIAL.ALARMS.CAM_START_JET_ANALISIS_CONNECTION_A;
END_REGION

REGION Network 22: UNIT 02 STATION 3 COAXIAL CAMERA START JET ANALISIS METHOD WORKING OR BLOCKED ALARM-------
   // CAMBIAR BIT DE DONE DEL METODO CORRECTO
   RUNG wire#powerrail
      Contact( "DB16201_METHODCALL_U01_STA3_MEAS_MEAS_NOOZLE_TRIGGER".Done )
      I_Contact( "DB16005_U02_STA3_COAXIAL_CLIENT_INTERFACE".U02_STA3_CAM_Method.TriggerStartCameraJetAnalisis.Outputs.Result )
      wire#w1
      Contact( "DB7257_UNIT_02_STA_3_COAXIAL_ENABLE_DISABLE".ENABLED )
      wire#w2
      Coil( "DB16000_OPC_UA_TRIGGER_ALARM".CLIENT.U02_STA3_COAXIAL.ALARMS.CAM_START_JET_ANALISIS_METHOD_WORKING_BLOCKED_A )
   END_RUNG
   RUNG wire#powerrail
      Contact( "DB16000_OPC_UA_TRIGGER_ALARM".CLIENT.U02_STA3_COAXIAL.ALARMS.CAM_START_JET_ANALISIS_METHOD_WORKING_BLOCKED_A )
      I_Contact( "DB2120_MPP_ITC_IPC".RESET_FAULTS )
   END_RUNG wire#w1
   RUNG wire#w2
      Coil( "DB426_ALARMS_WARNINGS".UNIT_01.OTHER."716601" )
   END_RUNG
   // the same network as SCL:
   "DB16000_OPC_UA_TRIGGER_ALARM".CLIENT.U02_STA3_COAXIAL.ALARMS.CAM_START_JET_ANALISIS_METHOD_WORKING_BLOCKED_A := (("DB16201_METHODCALL_U01_STA3_MEAS_MEAS_NOOZLE_TRIGGER".Done AND NOT "DB16005_U02_STA3_COAXIAL_CLIENT_INTERFACE".U02_STA3_CAM_Method.TriggerStartCameraJetAnalisis.Outputs.Result) OR ("DB16000_OPC_UA_TRIGGER_ALARM".CLIENT.U02_STA3_COAXIAL.ALARMS.CAM_START_JET_ANALISIS_METHOD_WORKING_BLOCKED_A AND NOT "DB2120_MPP_ITC_IPC".RESET_FAULTS)) AND "DB7257_UNIT_02_STA_3_COAXIAL_ENABLE_DISABLE".ENABLED;
   "DB426_ALARMS_WARNINGS".UNIT_01.OTHER."716601" := "DB16000_OPC_UA_TRIGGER_ALARM".CLIENT.U02_STA3_COAXIAL.ALARMS.CAM_START_JET_ANALISIS_METHOD_WORKING_BLOCKED_A;
END_REGION

REGION Network 23: UNIT 02 STATION 3 COAXIAL CAMERA START CLADDING ANALISIS METHOD CONNECTION ALARM ----------
   // CAMBIAR BIT DE ERROR DEL METODO CORRECTO
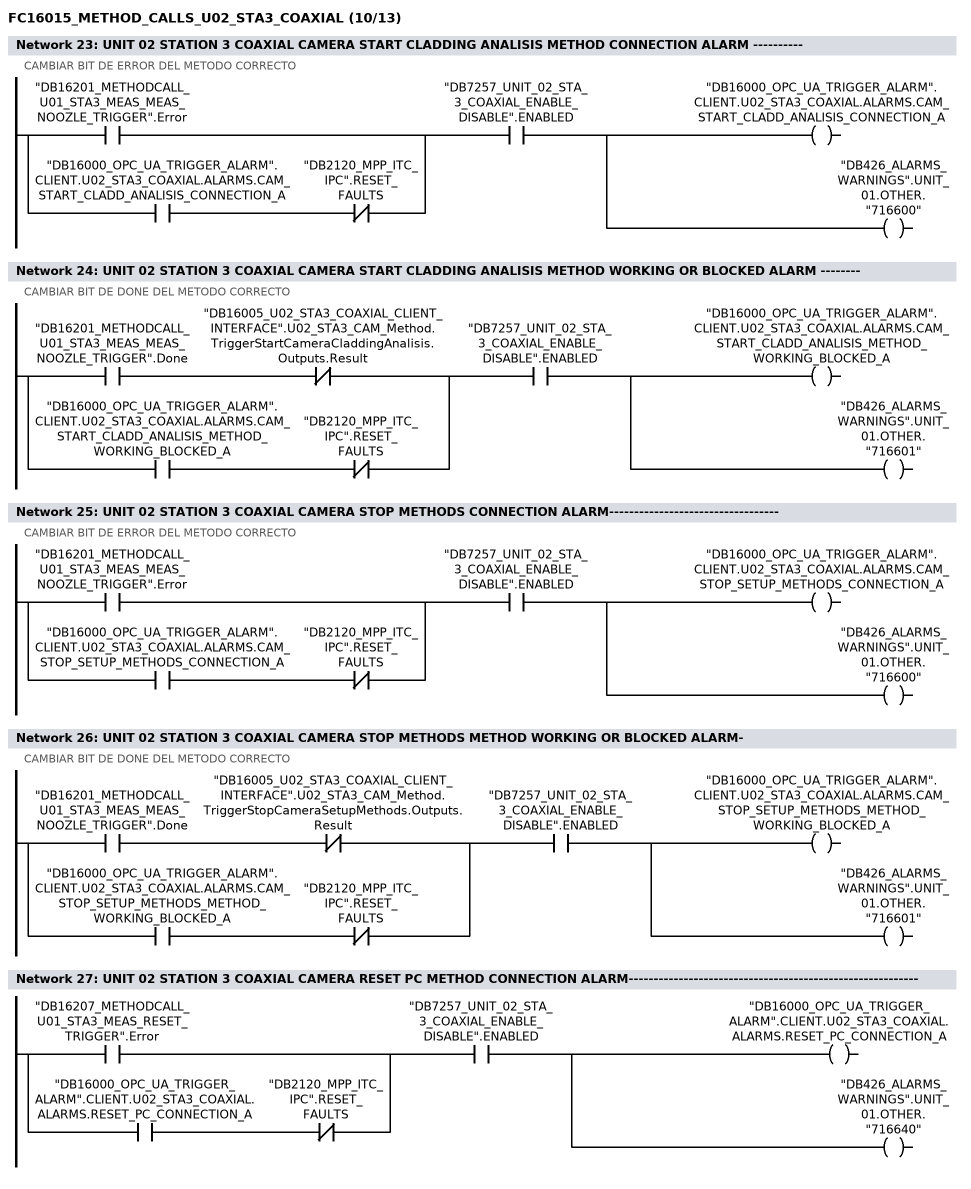
   RUNG wire#powerrail
      Contact( "DB16201_METHODCALL_U01_STA3_MEAS_MEAS_NOOZLE_TRIGGER".Error )
      wire#w1
      Contact( "DB7257_UNIT_02_STA_3_COAXIAL_ENABLE_DISABLE".ENABLED )
      wire#w2
      Coil( "DB16000_OPC_UA_TRIGGER_ALARM".CLIENT.U02_STA3_COAXIAL.ALARMS.CAM_START_CLADD_ANALISIS_CONNECTION_A )
   END_RUNG
   RUNG wire#powerrail
      Contact( "DB16000_OPC_UA_TRIGGER_ALARM".CLIENT.U02_STA3_COAXIAL.ALARMS.CAM_START_CLADD_ANALISIS_CONNECTION_A )
      I_Contact( "DB2120_MPP_ITC_IPC".RESET_FAULTS )
   END_RUNG wire#w1
   RUNG wire#w2
      Coil( "DB426_ALARMS_WARNINGS".UNIT_01.OTHER."716600" )
   END_RUNG
   // the same network as SCL:
   "DB16000_OPC_UA_TRIGGER_ALARM".CLIENT.U02_STA3_COAXIAL.ALARMS.CAM_START_CLADD_ANALISIS_CONNECTION_A := ("DB16201_METHODCALL_U01_STA3_MEAS_MEAS_NOOZLE_TRIGGER".Error OR ("DB16000_OPC_UA_TRIGGER_ALARM".CLIENT.U02_STA3_COAXIAL.ALARMS.CAM_START_CLADD_ANALISIS_CONNECTION_A AND NOT "DB2120_MPP_ITC_IPC".RESET_FAULTS)) AND "DB7257_UNIT_02_STA_3_COAXIAL_ENABLE_DISABLE".ENABLED;
   "DB426_ALARMS_WARNINGS".UNIT_01.OTHER."716600" := "DB16000_OPC_UA_TRIGGER_ALARM".CLIENT.U02_STA3_COAXIAL.ALARMS.CAM_START_CLADD_ANALISIS_CONNECTION_A;
END_REGION

REGION Network 24: UNIT 02 STATION 3 COAXIAL CAMERA START CLADDING ANALISIS METHOD WORKING OR BLOCKED ALARM --------
   // CAMBIAR BIT DE DONE DEL METODO CORRECTO
   RUNG wire#powerrail
      Contact( "DB16201_METHODCALL_U01_STA3_MEAS_MEAS_NOOZLE_TRIGGER".Done )
      I_Contact( "DB16005_U02_STA3_COAXIAL_CLIENT_INTERFACE".U02_STA3_CAM_Method.TriggerStartCameraCladdingAnalisis.Outputs.Result )
      wire#w1
      Contact( "DB7257_UNIT_02_STA_3_COAXIAL_ENABLE_DISABLE".ENABLED )
      wire#w2
      Coil( "DB16000_OPC_UA_TRIGGER_ALARM".CLIENT.U02_STA3_COAXIAL.ALARMS.CAM_START_CLADD_ANALISIS_METHOD_WORKING_BLOCKED_A )
   END_RUNG
   RUNG wire#powerrail
      Contact( "DB16000_OPC_UA_TRIGGER_ALARM".CLIENT.U02_STA3_COAXIAL.ALARMS.CAM_START_CLADD_ANALISIS_METHOD_WORKING_BLOCKED_A )
      I_Contact( "DB2120_MPP_ITC_IPC".RESET_FAULTS )
   END_RUNG wire#w1
   RUNG wire#w2
      Coil( "DB426_ALARMS_WARNINGS".UNIT_01.OTHER."716601" )
   END_RUNG
   // the same network as SCL:
   "DB16000_OPC_UA_TRIGGER_ALARM".CLIENT.U02_STA3_COAXIAL.ALARMS.CAM_START_CLADD_ANALISIS_METHOD_WORKING_BLOCKED_A := (("DB16201_METHODCALL_U01_STA3_MEAS_MEAS_NOOZLE_TRIGGER".Done AND NOT "DB16005_U02_STA3_COAXIAL_CLIENT_INTERFACE".U02_STA3_CAM_Method.TriggerStartCameraCladdingAnalisis.Outputs.Result) OR ("DB16000_OPC_UA_TRIGGER_ALARM".CLIENT.U02_STA3_COAXIAL.ALARMS.CAM_START_CLADD_ANALISIS_METHOD_WORKING_BLOCKED_A AND NOT "DB2120_MPP_ITC_IPC".RESET_FAULTS)) AND "DB7257_UNIT_02_STA_3_COAXIAL_ENABLE_DISABLE".ENABLED;
   "DB426_ALARMS_WARNINGS".UNIT_01.OTHER."716601" := "DB16000_OPC_UA_TRIGGER_ALARM".CLIENT.U02_STA3_COAXIAL.ALARMS.CAM_START_CLADD_ANALISIS_METHOD_WORKING_BLOCKED_A;
END_REGION

REGION Network 25: UNIT 02 STATION 3 COAXIAL CAMERA STOP METHODS CONNECTION ALARM----------------------------------
   // CAMBIAR BIT DE ERROR DEL METODO CORRECTO
   RUNG wire#powerrail
      Contact( "DB16201_METHODCALL_U01_STA3_MEAS_MEAS_NOOZLE_TRIGGER".Error )
      wire#w1
      Contact( "DB7257_UNIT_02_STA_3_COAXIAL_ENABLE_DISABLE".ENABLED )
      wire#w2
      Coil( "DB16000_OPC_UA_TRIGGER_ALARM".CLIENT.U02_STA3_COAXIAL.ALARMS.CAM_STOP_SETUP_METHODS_CONNECTION_A )
   END_RUNG
   RUNG wire#powerrail
      Contact( "DB16000_OPC_UA_TRIGGER_ALARM".CLIENT.U02_STA3_COAXIAL.ALARMS.CAM_STOP_SETUP_METHODS_CONNECTION_A )
      I_Contact( "DB2120_MPP_ITC_IPC".RESET_FAULTS )
   END_RUNG wire#w1
   RUNG wire#w2
      Coil( "DB426_ALARMS_WARNINGS".UNIT_01.OTHER."716600" )
   END_RUNG
   // the same network as SCL:
   "DB16000_OPC_UA_TRIGGER_ALARM".CLIENT.U02_STA3_COAXIAL.ALARMS.CAM_STOP_SETUP_METHODS_CONNECTION_A := ("DB16201_METHODCALL_U01_STA3_MEAS_MEAS_NOOZLE_TRIGGER".Error OR ("DB16000_OPC_UA_TRIGGER_ALARM".CLIENT.U02_STA3_COAXIAL.ALARMS.CAM_STOP_SETUP_METHODS_CONNECTION_A AND NOT "DB2120_MPP_ITC_IPC".RESET_FAULTS)) AND "DB7257_UNIT_02_STA_3_COAXIAL_ENABLE_DISABLE".ENABLED;
   "DB426_ALARMS_WARNINGS".UNIT_01.OTHER."716600" := "DB16000_OPC_UA_TRIGGER_ALARM".CLIENT.U02_STA3_COAXIAL.ALARMS.CAM_STOP_SETUP_METHODS_CONNECTION_A;
END_REGION

REGION Network 26: UNIT 02 STATION 3 COAXIAL CAMERA STOP METHODS METHOD WORKING OR BLOCKED ALARM-
   // CAMBIAR BIT DE DONE DEL METODO CORRECTO
   RUNG wire#powerrail
      Contact( "DB16201_METHODCALL_U01_STA3_MEAS_MEAS_NOOZLE_TRIGGER".Done )
      I_Contact( "DB16005_U02_STA3_COAXIAL_CLIENT_INTERFACE".U02_STA3_CAM_Method.TriggerStopCameraSetupMethods.Outputs.Result )
      wire#w1
      Contact( "DB7257_UNIT_02_STA_3_COAXIAL_ENABLE_DISABLE".ENABLED )
      wire#w2
      Coil( "DB16000_OPC_UA_TRIGGER_ALARM".CLIENT.U02_STA3_COAXIAL.ALARMS.CAM_STOP_SETUP_METHODS_METHOD_WORKING_BLOCKED_A )
   END_RUNG
   RUNG wire#powerrail
      Contact( "DB16000_OPC_UA_TRIGGER_ALARM".CLIENT.U02_STA3_COAXIAL.ALARMS.CAM_STOP_SETUP_METHODS_METHOD_WORKING_BLOCKED_A )
      I_Contact( "DB2120_MPP_ITC_IPC".RESET_FAULTS )
   END_RUNG wire#w1
   RUNG wire#w2
      Coil( "DB426_ALARMS_WARNINGS".UNIT_01.OTHER."716601" )
   END_RUNG
   // the same network as SCL:
   "DB16000_OPC_UA_TRIGGER_ALARM".CLIENT.U02_STA3_COAXIAL.ALARMS.CAM_STOP_SETUP_METHODS_METHOD_WORKING_BLOCKED_A := (("DB16201_METHODCALL_U01_STA3_MEAS_MEAS_NOOZLE_TRIGGER".Done AND NOT "DB16005_U02_STA3_COAXIAL_CLIENT_INTERFACE".U02_STA3_CAM_Method.TriggerStopCameraSetupMethods.Outputs.Result) OR ("DB16000_OPC_UA_TRIGGER_ALARM".CLIENT.U02_STA3_COAXIAL.ALARMS.CAM_STOP_SETUP_METHODS_METHOD_WORKING_BLOCKED_A AND NOT "DB2120_MPP_ITC_IPC".RESET_FAULTS)) AND "DB7257_UNIT_02_STA_3_COAXIAL_ENABLE_DISABLE".ENABLED;
   "DB426_ALARMS_WARNINGS".UNIT_01.OTHER."716601" := "DB16000_OPC_UA_TRIGGER_ALARM".CLIENT.U02_STA3_COAXIAL.ALARMS.CAM_STOP_SETUP_METHODS_METHOD_WORKING_BLOCKED_A;
END_REGION

REGION Network 27: UNIT 02 STATION 3 COAXIAL CAMERA RESET PC METHOD CONNECTION ALARM----------------------------------------------------------
   RUNG wire#powerrail
      Contact( "DB16207_METHODCALL_U01_STA3_MEAS_RESET_TRIGGER".Error )
      wire#w1
      Contact( "DB7257_UNIT_02_STA_3_COAXIAL_ENABLE_DISABLE".ENABLED )
      wire#w2
      Coil( "DB16000_OPC_UA_TRIGGER_ALARM".CLIENT.U02_STA3_COAXIAL.ALARMS.RESET_PC_CONNECTION_A )
   END_RUNG
   RUNG wire#powerrail
      Contact( "DB16000_OPC_UA_TRIGGER_ALARM".CLIENT.U02_STA3_COAXIAL.ALARMS.RESET_PC_CONNECTION_A )
      I_Contact( "DB2120_MPP_ITC_IPC".RESET_FAULTS )
   END_RUNG wire#w1
   RUNG wire#w2
      Coil( "DB426_ALARMS_WARNINGS".UNIT_01.OTHER."716640" )
   END_RUNG
   // the same network as SCL:
   "DB16000_OPC_UA_TRIGGER_ALARM".CLIENT.U02_STA3_COAXIAL.ALARMS.RESET_PC_CONNECTION_A := ("DB16207_METHODCALL_U01_STA3_MEAS_RESET_TRIGGER".Error OR ("DB16000_OPC_UA_TRIGGER_ALARM".CLIENT.U02_STA3_COAXIAL.ALARMS.RESET_PC_CONNECTION_A AND NOT "DB2120_MPP_ITC_IPC".RESET_FAULTS)) AND "DB7257_UNIT_02_STA_3_COAXIAL_ENABLE_DISABLE".ENABLED;
   "DB426_ALARMS_WARNINGS".UNIT_01.OTHER."716640" := "DB16000_OPC_UA_TRIGGER_ALARM".CLIENT.U02_STA3_COAXIAL.ALARMS.RESET_PC_CONNECTION_A;
END_REGION

REGION Network 28: UNIT 02 STATION 3 COAXIAL CAMERA RESET PC METHOD WORKING OR BLOCKED ALARM-----------------------------------------
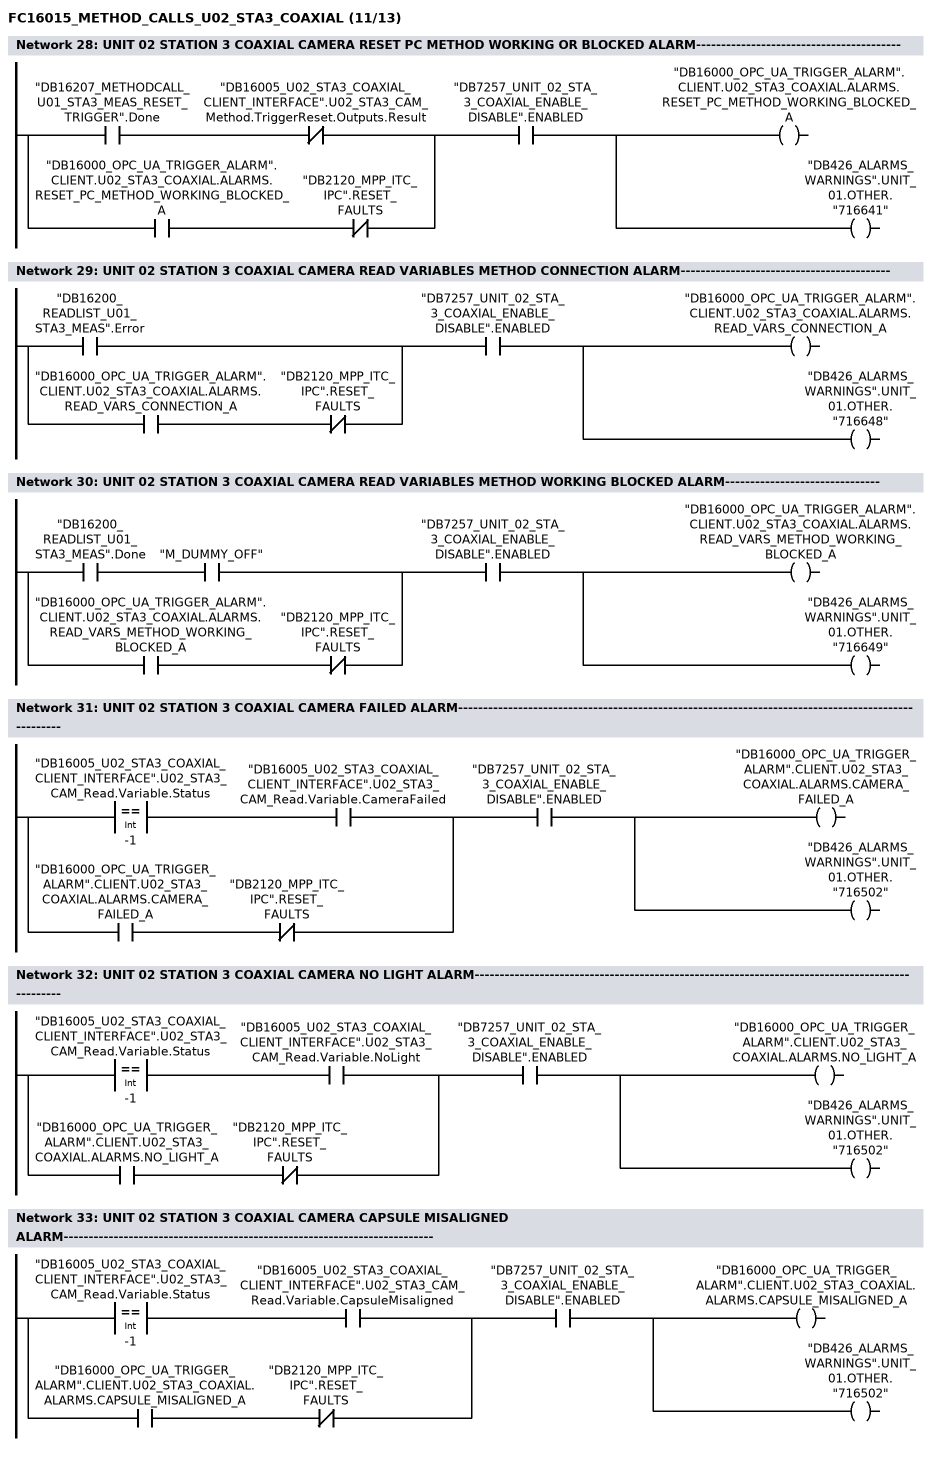
   RUNG wire#powerrail
      Contact( "DB16207_METHODCALL_U01_STA3_MEAS_RESET_TRIGGER".Done )
      I_Contact( "DB16005_U02_STA3_COAXIAL_CLIENT_INTERFACE".U02_STA3_CAM_Method.TriggerReset.Outputs.Result )
      wire#w1
      Contact( "DB7257_UNIT_02_STA_3_COAXIAL_ENABLE_DISABLE".ENABLED )
      wire#w2
      Coil( "DB16000_OPC_UA_TRIGGER_ALARM".CLIENT.U02_STA3_COAXIAL.ALARMS.RESET_PC_METHOD_WORKING_BLOCKED_A )
   END_RUNG
   RUNG wire#powerrail
      Contact( "DB16000_OPC_UA_TRIGGER_ALARM".CLIENT.U02_STA3_COAXIAL.ALARMS.RESET_PC_METHOD_WORKING_BLOCKED_A )
      I_Contact( "DB2120_MPP_ITC_IPC".RESET_FAULTS )
   END_RUNG wire#w1
   RUNG wire#w2
      Coil( "DB426_ALARMS_WARNINGS".UNIT_01.OTHER."716641" )
   END_RUNG
   // the same network as SCL:
   "DB16000_OPC_UA_TRIGGER_ALARM".CLIENT.U02_STA3_COAXIAL.ALARMS.RESET_PC_METHOD_WORKING_BLOCKED_A := (("DB16207_METHODCALL_U01_STA3_MEAS_RESET_TRIGGER".Done AND NOT "DB16005_U02_STA3_COAXIAL_CLIENT_INTERFACE".U02_STA3_CAM_Method.TriggerReset.Outputs.Result) OR ("DB16000_OPC_UA_TRIGGER_ALARM".CLIENT.U02_STA3_COAXIAL.ALARMS.RESET_PC_METHOD_WORKING_BLOCKED_A AND NOT "DB2120_MPP_ITC_IPC".RESET_FAULTS)) AND "DB7257_UNIT_02_STA_3_COAXIAL_ENABLE_DISABLE".ENABLED;
   "DB426_ALARMS_WARNINGS".UNIT_01.OTHER."716641" := "DB16000_OPC_UA_TRIGGER_ALARM".CLIENT.U02_STA3_COAXIAL.ALARMS.RESET_PC_METHOD_WORKING_BLOCKED_A;
END_REGION

REGION Network 29: UNIT 02 STATION 3 COAXIAL CAMERA READ VARIABLES METHOD CONNECTION ALARM------------------------------------------
   RUNG wire#powerrail
      Contact( "DB16200_READLIST_U01_STA3_MEAS".Error )
      wire#w1
      Contact( "DB7257_UNIT_02_STA_3_COAXIAL_ENABLE_DISABLE".ENABLED )
      wire#w2
      Coil( "DB16000_OPC_UA_TRIGGER_ALARM".CLIENT.U02_STA3_COAXIAL.ALARMS.READ_VARS_CONNECTION_A )
   END_RUNG
   RUNG wire#powerrail
      Contact( "DB16000_OPC_UA_TRIGGER_ALARM".CLIENT.U02_STA3_COAXIAL.ALARMS.READ_VARS_CONNECTION_A )
      I_Contact( "DB2120_MPP_ITC_IPC".RESET_FAULTS )
   END_RUNG wire#w1
   RUNG wire#w2
      Coil( "DB426_ALARMS_WARNINGS".UNIT_01.OTHER."716648" )
   END_RUNG
   // the same network as SCL:
   "DB16000_OPC_UA_TRIGGER_ALARM".CLIENT.U02_STA3_COAXIAL.ALARMS.READ_VARS_CONNECTION_A := ("DB16200_READLIST_U01_STA3_MEAS".Error OR ("DB16000_OPC_UA_TRIGGER_ALARM".CLIENT.U02_STA3_COAXIAL.ALARMS.READ_VARS_CONNECTION_A AND NOT "DB2120_MPP_ITC_IPC".RESET_FAULTS)) AND "DB7257_UNIT_02_STA_3_COAXIAL_ENABLE_DISABLE".ENABLED;
   "DB426_ALARMS_WARNINGS".UNIT_01.OTHER."716648" := "DB16000_OPC_UA_TRIGGER_ALARM".CLIENT.U02_STA3_COAXIAL.ALARMS.READ_VARS_CONNECTION_A;
END_REGION

REGION Network 30: UNIT 02 STATION 3 COAXIAL CAMERA READ VARIABLES METHOD WORKING BLOCKED ALARM-------------------------------
   RUNG wire#powerrail
      Contact( "DB16200_READLIST_U01_STA3_MEAS".Done )
      Contact( "M_DUMMY_OFF" )
      wire#w1
      Contact( "DB7257_UNIT_02_STA_3_COAXIAL_ENABLE_DISABLE".ENABLED )
      wire#w2
      Coil( "DB16000_OPC_UA_TRIGGER_ALARM".CLIENT.U02_STA3_COAXIAL.ALARMS.READ_VARS_METHOD_WORKING_BLOCKED_A )
   END_RUNG
   RUNG wire#powerrail
      Contact( "DB16000_OPC_UA_TRIGGER_ALARM".CLIENT.U02_STA3_COAXIAL.ALARMS.READ_VARS_METHOD_WORKING_BLOCKED_A )
      I_Contact( "DB2120_MPP_ITC_IPC".RESET_FAULTS )
   END_RUNG wire#w1
   RUNG wire#w2
      Coil( "DB426_ALARMS_WARNINGS".UNIT_01.OTHER."716649" )
   END_RUNG
   // the same network as SCL:
   "DB16000_OPC_UA_TRIGGER_ALARM".CLIENT.U02_STA3_COAXIAL.ALARMS.READ_VARS_METHOD_WORKING_BLOCKED_A := (("DB16200_READLIST_U01_STA3_MEAS".Done AND "M_DUMMY_OFF") OR ("DB16000_OPC_UA_TRIGGER_ALARM".CLIENT.U02_STA3_COAXIAL.ALARMS.READ_VARS_METHOD_WORKING_BLOCKED_A AND NOT "DB2120_MPP_ITC_IPC".RESET_FAULTS)) AND "DB7257_UNIT_02_STA_3_COAXIAL_ENABLE_DISABLE".ENABLED;
   "DB426_ALARMS_WARNINGS".UNIT_01.OTHER."716649" := "DB16000_OPC_UA_TRIGGER_ALARM".CLIENT.U02_STA3_COAXIAL.ALARMS.READ_VARS_METHOD_WORKING_BLOCKED_A;
END_REGION

REGION Network 31: UNIT 02 STATION 3 COAXIAL CAMERA FAILED ALARM----------------------------------------------------------------------------------------------------
   RUNG wire#powerrail
      { S7_Templates := "SrcType := Int" } EQ_Contact(in1 := "DB16005_U02_STA3_COAXIAL_CLIENT_INTERFACE".U02_STA3_CAM_Read.Variable.Status, in2 := -1)
      Contact( "DB16005_U02_STA3_COAXIAL_CLIENT_INTERFACE".U02_STA3_CAM_Read.Variable.CameraFailed )
      wire#w1
      Contact( "DB7257_UNIT_02_STA_3_COAXIAL_ENABLE_DISABLE".ENABLED )
      wire#w2
      Coil( "DB16000_OPC_UA_TRIGGER_ALARM".CLIENT.U02_STA3_COAXIAL.ALARMS.CAMERA_FAILED_A )
   END_RUNG
   RUNG wire#powerrail
      Contact( "DB16000_OPC_UA_TRIGGER_ALARM".CLIENT.U02_STA3_COAXIAL.ALARMS.CAMERA_FAILED_A )
      I_Contact( "DB2120_MPP_ITC_IPC".RESET_FAULTS )
   END_RUNG wire#w1
   RUNG wire#w2
      Coil( "DB426_ALARMS_WARNINGS".UNIT_01.OTHER."716502" )
   END_RUNG
   // the same network as SCL:
   "DB16000_OPC_UA_TRIGGER_ALARM".CLIENT.U02_STA3_COAXIAL.ALARMS.CAMERA_FAILED_A := ((("DB16005_U02_STA3_COAXIAL_CLIENT_INTERFACE".U02_STA3_CAM_Read.Variable.Status = (-1)) AND "DB16005_U02_STA3_COAXIAL_CLIENT_INTERFACE".U02_STA3_CAM_Read.Variable.CameraFailed) OR ("DB16000_OPC_UA_TRIGGER_ALARM".CLIENT.U02_STA3_COAXIAL.ALARMS.CAMERA_FAILED_A AND NOT "DB2120_MPP_ITC_IPC".RESET_FAULTS)) AND "DB7257_UNIT_02_STA_3_COAXIAL_ENABLE_DISABLE".ENABLED;
   "DB426_ALARMS_WARNINGS".UNIT_01.OTHER."716502" := "DB16000_OPC_UA_TRIGGER_ALARM".CLIENT.U02_STA3_COAXIAL.ALARMS.CAMERA_FAILED_A;
END_REGION

REGION Network 32: UNIT 02 STATION 3 COAXIAL CAMERA NO LIGHT ALARM------------------------------------------------------------------------------------------------
   RUNG wire#powerrail
      { S7_Templates := "SrcType := Int" } EQ_Contact(in1 := "DB16005_U02_STA3_COAXIAL_CLIENT_INTERFACE".U02_STA3_CAM_Read.Variable.Status, in2 := -1)
      Contact( "DB16005_U02_STA3_COAXIAL_CLIENT_INTERFACE".U02_STA3_CAM_Read.Variable.NoLight )
      wire#w1
      Contact( "DB7257_UNIT_02_STA_3_COAXIAL_ENABLE_DISABLE".ENABLED )
      wire#w2
      Coil( "DB16000_OPC_UA_TRIGGER_ALARM".CLIENT.U02_STA3_COAXIAL.ALARMS.NO_LIGHT_A )
   END_RUNG
   RUNG wire#powerrail
      Contact( "DB16000_OPC_UA_TRIGGER_ALARM".CLIENT.U02_STA3_COAXIAL.ALARMS.NO_LIGHT_A )
      I_Contact( "DB2120_MPP_ITC_IPC".RESET_FAULTS )
   END_RUNG wire#w1
   RUNG wire#w2
      Coil( "DB426_ALARMS_WARNINGS".UNIT_01.OTHER."716502" )
   END_RUNG
   // the same network as SCL:
   "DB16000_OPC_UA_TRIGGER_ALARM".CLIENT.U02_STA3_COAXIAL.ALARMS.NO_LIGHT_A := ((("DB16005_U02_STA3_COAXIAL_CLIENT_INTERFACE".U02_STA3_CAM_Read.Variable.Status = (-1)) AND "DB16005_U02_STA3_COAXIAL_CLIENT_INTERFACE".U02_STA3_CAM_Read.Variable.NoLight) OR ("DB16000_OPC_UA_TRIGGER_ALARM".CLIENT.U02_STA3_COAXIAL.ALARMS.NO_LIGHT_A AND NOT "DB2120_MPP_ITC_IPC".RESET_FAULTS)) AND "DB7257_UNIT_02_STA_3_COAXIAL_ENABLE_DISABLE".ENABLED;
   "DB426_ALARMS_WARNINGS".UNIT_01.OTHER."716502" := "DB16000_OPC_UA_TRIGGER_ALARM".CLIENT.U02_STA3_COAXIAL.ALARMS.NO_LIGHT_A;
END_REGION

REGION Network 33: UNIT 02 STATION 3 COAXIAL CAMERA CAPSULE MISALIGNED ALARM--------------------------------------------------------------------------
   RUNG wire#powerrail
      { S7_Templates := "SrcType := Int" } EQ_Contact(in1 := "DB16005_U02_STA3_COAXIAL_CLIENT_INTERFACE".U02_STA3_CAM_Read.Variable.Status, in2 := -1)
      Contact( "DB16005_U02_STA3_COAXIAL_CLIENT_INTERFACE".U02_STA3_CAM_Read.Variable.CapsuleMisaligned )
      wire#w1
      Contact( "DB7257_UNIT_02_STA_3_COAXIAL_ENABLE_DISABLE".ENABLED )
      wire#w2
      Coil( "DB16000_OPC_UA_TRIGGER_ALARM".CLIENT.U02_STA3_COAXIAL.ALARMS.CAPSULE_MISALIGNED_A )
   END_RUNG
   RUNG wire#powerrail
      Contact( "DB16000_OPC_UA_TRIGGER_ALARM".CLIENT.U02_STA3_COAXIAL.ALARMS.CAPSULE_MISALIGNED_A )
      I_Contact( "DB2120_MPP_ITC_IPC".RESET_FAULTS )
   END_RUNG wire#w1
   RUNG wire#w2
      Coil( "DB426_ALARMS_WARNINGS".UNIT_01.OTHER."716502" )
   END_RUNG
   // the same network as SCL:
   "DB16000_OPC_UA_TRIGGER_ALARM".CLIENT.U02_STA3_COAXIAL.ALARMS.CAPSULE_MISALIGNED_A := ((("DB16005_U02_STA3_COAXIAL_CLIENT_INTERFACE".U02_STA3_CAM_Read.Variable.Status = (-1)) AND "DB16005_U02_STA3_COAXIAL_CLIENT_INTERFACE".U02_STA3_CAM_Read.Variable.CapsuleMisaligned) OR ("DB16000_OPC_UA_TRIGGER_ALARM".CLIENT.U02_STA3_COAXIAL.ALARMS.CAPSULE_MISALIGNED_A AND NOT "DB2120_MPP_ITC_IPC".RESET_FAULTS)) AND "DB7257_UNIT_02_STA_3_COAXIAL_ENABLE_DISABLE".ENABLED;
   "DB426_ALARMS_WARNINGS".UNIT_01.OTHER."716502" := "DB16000_OPC_UA_TRIGGER_ALARM".CLIENT.U02_STA3_COAXIAL.ALARMS.CAPSULE_MISALIGNED_A;
END_REGION

REGION Network 34: UNIT 02 STATION 3 COAXIAL CAMERA JET FAILED ALARM-----------------------------------------------------------------------------------------------
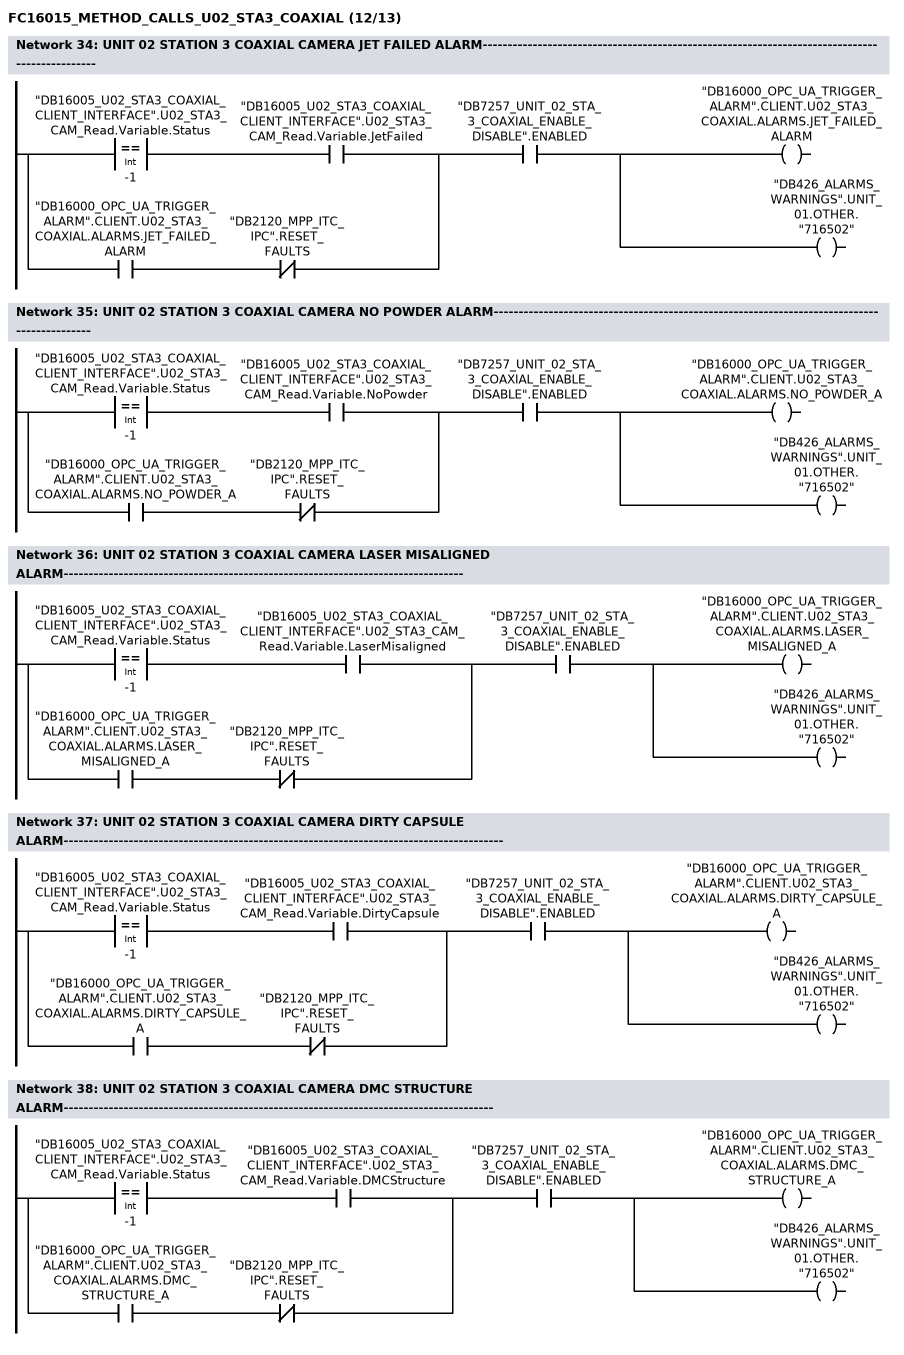
   RUNG wire#powerrail
      { S7_Templates := "SrcType := Int" } EQ_Contact(in1 := "DB16005_U02_STA3_COAXIAL_CLIENT_INTERFACE".U02_STA3_CAM_Read.Variable.Status, in2 := -1)
      Contact( "DB16005_U02_STA3_COAXIAL_CLIENT_INTERFACE".U02_STA3_CAM_Read.Variable.JetFailed )
      wire#w1
      Contact( "DB7257_UNIT_02_STA_3_COAXIAL_ENABLE_DISABLE".ENABLED )
      wire#w2
      Coil( "DB16000_OPC_UA_TRIGGER_ALARM".CLIENT.U02_STA3_COAXIAL.ALARMS.JET_FAILED_ALARM )
   END_RUNG
   RUNG wire#powerrail
      Contact( "DB16000_OPC_UA_TRIGGER_ALARM".CLIENT.U02_STA3_COAXIAL.ALARMS.JET_FAILED_ALARM )
      I_Contact( "DB2120_MPP_ITC_IPC".RESET_FAULTS )
   END_RUNG wire#w1
   RUNG wire#w2
      Coil( "DB426_ALARMS_WARNINGS".UNIT_01.OTHER."716502" )
   END_RUNG
   // the same network as SCL:
   "DB16000_OPC_UA_TRIGGER_ALARM".CLIENT.U02_STA3_COAXIAL.ALARMS.JET_FAILED_ALARM := ((("DB16005_U02_STA3_COAXIAL_CLIENT_INTERFACE".U02_STA3_CAM_Read.Variable.Status = (-1)) AND "DB16005_U02_STA3_COAXIAL_CLIENT_INTERFACE".U02_STA3_CAM_Read.Variable.JetFailed) OR ("DB16000_OPC_UA_TRIGGER_ALARM".CLIENT.U02_STA3_COAXIAL.ALARMS.JET_FAILED_ALARM AND NOT "DB2120_MPP_ITC_IPC".RESET_FAULTS)) AND "DB7257_UNIT_02_STA_3_COAXIAL_ENABLE_DISABLE".ENABLED;
   "DB426_ALARMS_WARNINGS".UNIT_01.OTHER."716502" := "DB16000_OPC_UA_TRIGGER_ALARM".CLIENT.U02_STA3_COAXIAL.ALARMS.JET_FAILED_ALARM;
END_REGION

REGION Network 35: UNIT 02 STATION 3 COAXIAL CAMERA NO POWDER ALARM--------------------------------------------------------------------------------------------
   RUNG wire#powerrail
      { S7_Templates := "SrcType := Int" } EQ_Contact(in1 := "DB16005_U02_STA3_COAXIAL_CLIENT_INTERFACE".U02_STA3_CAM_Read.Variable.Status, in2 := -1)
      Contact( "DB16005_U02_STA3_COAXIAL_CLIENT_INTERFACE".U02_STA3_CAM_Read.Variable.NoPowder )
      wire#w1
      Contact( "DB7257_UNIT_02_STA_3_COAXIAL_ENABLE_DISABLE".ENABLED )
      wire#w2
      Coil( "DB16000_OPC_UA_TRIGGER_ALARM".CLIENT.U02_STA3_COAXIAL.ALARMS.NO_POWDER_A )
   END_RUNG
   RUNG wire#powerrail
      Contact( "DB16000_OPC_UA_TRIGGER_ALARM".CLIENT.U02_STA3_COAXIAL.ALARMS.NO_POWDER_A )
      I_Contact( "DB2120_MPP_ITC_IPC".RESET_FAULTS )
   END_RUNG wire#w1
   RUNG wire#w2
      Coil( "DB426_ALARMS_WARNINGS".UNIT_01.OTHER."716502" )
   END_RUNG
   // the same network as SCL:
   "DB16000_OPC_UA_TRIGGER_ALARM".CLIENT.U02_STA3_COAXIAL.ALARMS.NO_POWDER_A := ((("DB16005_U02_STA3_COAXIAL_CLIENT_INTERFACE".U02_STA3_CAM_Read.Variable.Status = (-1)) AND "DB16005_U02_STA3_COAXIAL_CLIENT_INTERFACE".U02_STA3_CAM_Read.Variable.NoPowder) OR ("DB16000_OPC_UA_TRIGGER_ALARM".CLIENT.U02_STA3_COAXIAL.ALARMS.NO_POWDER_A AND NOT "DB2120_MPP_ITC_IPC".RESET_FAULTS)) AND "DB7257_UNIT_02_STA_3_COAXIAL_ENABLE_DISABLE".ENABLED;
   "DB426_ALARMS_WARNINGS".UNIT_01.OTHER."716502" := "DB16000_OPC_UA_TRIGGER_ALARM".CLIENT.U02_STA3_COAXIAL.ALARMS.NO_POWDER_A;
END_REGION

REGION Network 36: UNIT 02 STATION 3 COAXIAL CAMERA LASER MISALIGNED ALARM--------------------------------------------------------------------------------
   RUNG wire#powerrail
      { S7_Templates := "SrcType := Int" } EQ_Contact(in1 := "DB16005_U02_STA3_COAXIAL_CLIENT_INTERFACE".U02_STA3_CAM_Read.Variable.Status, in2 := -1)
      Contact( "DB16005_U02_STA3_COAXIAL_CLIENT_INTERFACE".U02_STA3_CAM_Read.Variable.LaserMisaligned )
      wire#w1
      Contact( "DB7257_UNIT_02_STA_3_COAXIAL_ENABLE_DISABLE".ENABLED )
      wire#w2
      Coil( "DB16000_OPC_UA_TRIGGER_ALARM".CLIENT.U02_STA3_COAXIAL.ALARMS.LASER_MISALIGNED_A )
   END_RUNG
   RUNG wire#powerrail
      Contact( "DB16000_OPC_UA_TRIGGER_ALARM".CLIENT.U02_STA3_COAXIAL.ALARMS.LASER_MISALIGNED_A )
      I_Contact( "DB2120_MPP_ITC_IPC".RESET_FAULTS )
   END_RUNG wire#w1
   RUNG wire#w2
      Coil( "DB426_ALARMS_WARNINGS".UNIT_01.OTHER."716502" )
   END_RUNG
   // the same network as SCL:
   "DB16000_OPC_UA_TRIGGER_ALARM".CLIENT.U02_STA3_COAXIAL.ALARMS.LASER_MISALIGNED_A := ((("DB16005_U02_STA3_COAXIAL_CLIENT_INTERFACE".U02_STA3_CAM_Read.Variable.Status = (-1)) AND "DB16005_U02_STA3_COAXIAL_CLIENT_INTERFACE".U02_STA3_CAM_Read.Variable.LaserMisaligned) OR ("DB16000_OPC_UA_TRIGGER_ALARM".CLIENT.U02_STA3_COAXIAL.ALARMS.LASER_MISALIGNED_A AND NOT "DB2120_MPP_ITC_IPC".RESET_FAULTS)) AND "DB7257_UNIT_02_STA_3_COAXIAL_ENABLE_DISABLE".ENABLED;
   "DB426_ALARMS_WARNINGS".UNIT_01.OTHER."716502" := "DB16000_OPC_UA_TRIGGER_ALARM".CLIENT.U02_STA3_COAXIAL.ALARMS.LASER_MISALIGNED_A;
END_REGION

REGION Network 37: UNIT 02 STATION 3 COAXIAL CAMERA DIRTY CAPSULE ALARM----------------------------------------------------------------------------------------
   RUNG wire#powerrail
      { S7_Templates := "SrcType := Int" } EQ_Contact(in1 := "DB16005_U02_STA3_COAXIAL_CLIENT_INTERFACE".U02_STA3_CAM_Read.Variable.Status, in2 := -1)
      Contact( "DB16005_U02_STA3_COAXIAL_CLIENT_INTERFACE".U02_STA3_CAM_Read.Variable.DirtyCapsule )
      wire#w1
      Contact( "DB7257_UNIT_02_STA_3_COAXIAL_ENABLE_DISABLE".ENABLED )
      wire#w2
      Coil( "DB16000_OPC_UA_TRIGGER_ALARM".CLIENT.U02_STA3_COAXIAL.ALARMS.DIRTY_CAPSULE_A )
   END_RUNG
   RUNG wire#powerrail
      Contact( "DB16000_OPC_UA_TRIGGER_ALARM".CLIENT.U02_STA3_COAXIAL.ALARMS.DIRTY_CAPSULE_A )
      I_Contact( "DB2120_MPP_ITC_IPC".RESET_FAULTS )
   END_RUNG wire#w1
   RUNG wire#w2
      Coil( "DB426_ALARMS_WARNINGS".UNIT_01.OTHER."716502" )
   END_RUNG
   // the same network as SCL:
   "DB16000_OPC_UA_TRIGGER_ALARM".CLIENT.U02_STA3_COAXIAL.ALARMS.DIRTY_CAPSULE_A := ((("DB16005_U02_STA3_COAXIAL_CLIENT_INTERFACE".U02_STA3_CAM_Read.Variable.Status = (-1)) AND "DB16005_U02_STA3_COAXIAL_CLIENT_INTERFACE".U02_STA3_CAM_Read.Variable.DirtyCapsule) OR ("DB16000_OPC_UA_TRIGGER_ALARM".CLIENT.U02_STA3_COAXIAL.ALARMS.DIRTY_CAPSULE_A AND NOT "DB2120_MPP_ITC_IPC".RESET_FAULTS)) AND "DB7257_UNIT_02_STA_3_COAXIAL_ENABLE_DISABLE".ENABLED;
   "DB426_ALARMS_WARNINGS".UNIT_01.OTHER."716502" := "DB16000_OPC_UA_TRIGGER_ALARM".CLIENT.U02_STA3_COAXIAL.ALARMS.DIRTY_CAPSULE_A;
END_REGION

REGION Network 38: UNIT 02 STATION 3 COAXIAL CAMERA DMC STRUCTURE ALARM--------------------------------------------------------------------------------------
   RUNG wire#powerrail
      { S7_Templates := "SrcType := Int" } EQ_Contact(in1 := "DB16005_U02_STA3_COAXIAL_CLIENT_INTERFACE".U02_STA3_CAM_Read.Variable.Status, in2 := -1)
      Contact( "DB16005_U02_STA3_COAXIAL_CLIENT_INTERFACE".U02_STA3_CAM_Read.Variable.DMCStructure )
      wire#w1
      Contact( "DB7257_UNIT_02_STA_3_COAXIAL_ENABLE_DISABLE".ENABLED )
      wire#w2
      Coil( "DB16000_OPC_UA_TRIGGER_ALARM".CLIENT.U02_STA3_COAXIAL.ALARMS.DMC_STRUCTURE_A )
   END_RUNG
   RUNG wire#powerrail
      Contact( "DB16000_OPC_UA_TRIGGER_ALARM".CLIENT.U02_STA3_COAXIAL.ALARMS.DMC_STRUCTURE_A )
      I_Contact( "DB2120_MPP_ITC_IPC".RESET_FAULTS )
   END_RUNG wire#w1
   RUNG wire#w2
      Coil( "DB426_ALARMS_WARNINGS".UNIT_01.OTHER."716502" )
   END_RUNG
   // the same network as SCL:
   "DB16000_OPC_UA_TRIGGER_ALARM".CLIENT.U02_STA3_COAXIAL.ALARMS.DMC_STRUCTURE_A := ((("DB16005_U02_STA3_COAXIAL_CLIENT_INTERFACE".U02_STA3_CAM_Read.Variable.Status = (-1)) AND "DB16005_U02_STA3_COAXIAL_CLIENT_INTERFACE".U02_STA3_CAM_Read.Variable.DMCStructure) OR ("DB16000_OPC_UA_TRIGGER_ALARM".CLIENT.U02_STA3_COAXIAL.ALARMS.DMC_STRUCTURE_A AND NOT "DB2120_MPP_ITC_IPC".RESET_FAULTS)) AND "DB7257_UNIT_02_STA_3_COAXIAL_ENABLE_DISABLE".ENABLED;
   "DB426_ALARMS_WARNINGS".UNIT_01.OTHER."716502" := "DB16000_OPC_UA_TRIGGER_ALARM".CLIENT.U02_STA3_COAXIAL.ALARMS.DMC_STRUCTURE_A;
END_REGION

REGION Network 39: IS_SEOC ALARMS
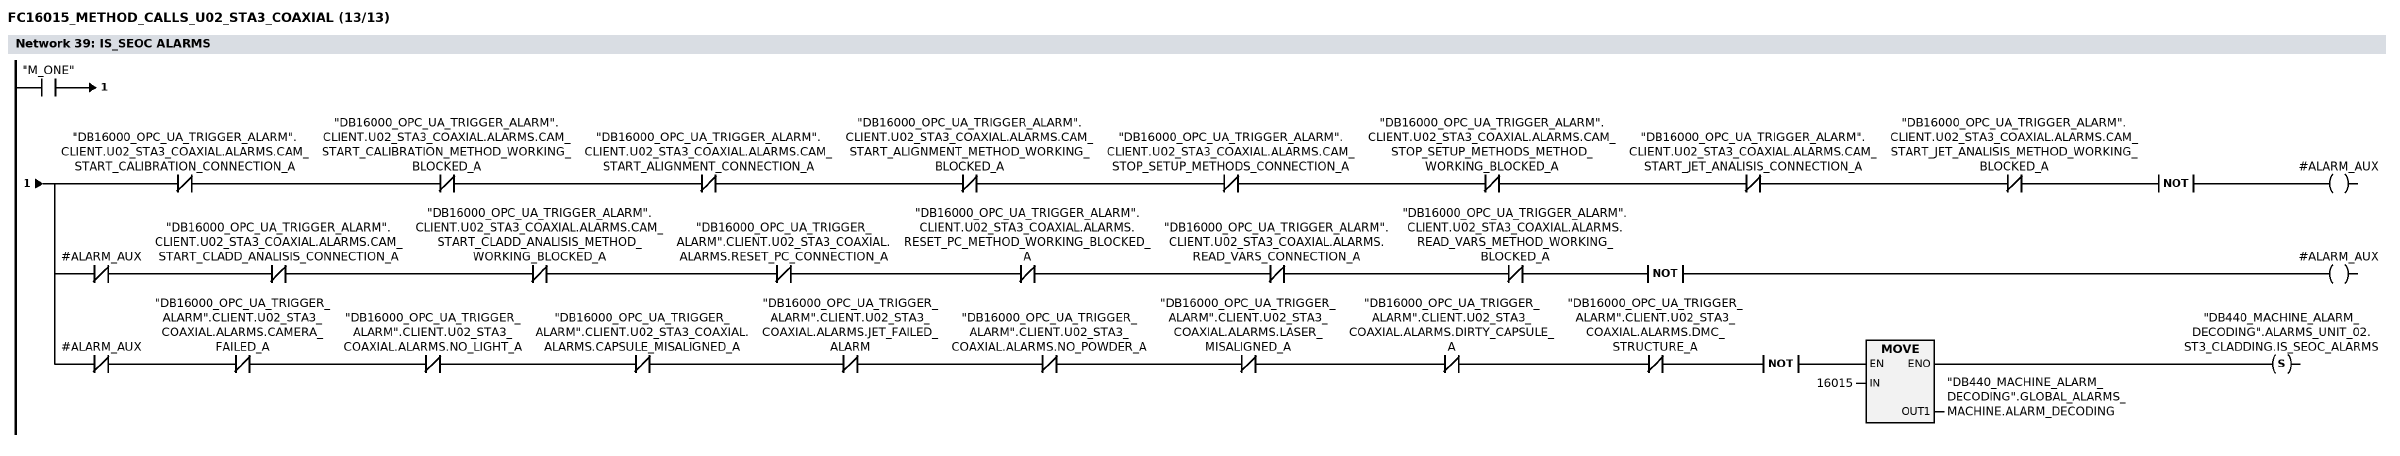
   RUNG wire#powerrail
      Contact( "M_ONE" )
      wire#w1
      I_Contact( "DB16000_OPC_UA_TRIGGER_ALARM".CLIENT.U02_STA3_COAXIAL.ALARMS.CAM_START_CALIBRATION_CONNECTION_A )
      I_Contact( "DB16000_OPC_UA_TRIGGER_ALARM".CLIENT.U02_STA3_COAXIAL.ALARMS.CAM_START_CALIBRATION_METHOD_WORKING_BLOCKED_A )
      I_Contact( "DB16000_OPC_UA_TRIGGER_ALARM".CLIENT.U02_STA3_COAXIAL.ALARMS.CAM_START_ALIGNMENT_CONNECTION_A )
      I_Contact( "DB16000_OPC_UA_TRIGGER_ALARM".CLIENT.U02_STA3_COAXIAL.ALARMS.CAM_START_ALIGNMENT_METHOD_WORKING_BLOCKED_A )
      I_Contact( "DB16000_OPC_UA_TRIGGER_ALARM".CLIENT.U02_STA3_COAXIAL.ALARMS.CAM_STOP_SETUP_METHODS_CONNECTION_A )
      I_Contact( "DB16000_OPC_UA_TRIGGER_ALARM".CLIENT.U02_STA3_COAXIAL.ALARMS.CAM_STOP_SETUP_METHODS_METHOD_WORKING_BLOCKED_A )
      I_Contact( "DB16000_OPC_UA_TRIGGER_ALARM".CLIENT.U02_STA3_COAXIAL.ALARMS.CAM_START_JET_ANALISIS_CONNECTION_A )
      I_Contact( "DB16000_OPC_UA_TRIGGER_ALARM".CLIENT.U02_STA3_COAXIAL.ALARMS.CAM_START_JET_ANALISIS_METHOD_WORKING_BLOCKED_A )
      Not()
      Coil( #ALARM_AUX )
   END_RUNG
   RUNG wire#w1
      I_Contact( #ALARM_AUX )
      I_Contact( "DB16000_OPC_UA_TRIGGER_ALARM".CLIENT.U02_STA3_COAXIAL.ALARMS.CAM_START_CLADD_ANALISIS_CONNECTION_A )
      I_Contact( "DB16000_OPC_UA_TRIGGER_ALARM".CLIENT.U02_STA3_COAXIAL.ALARMS.CAM_START_CLADD_ANALISIS_METHOD_WORKING_BLOCKED_A )
      I_Contact( "DB16000_OPC_UA_TRIGGER_ALARM".CLIENT.U02_STA3_COAXIAL.ALARMS.RESET_PC_CONNECTION_A )
      I_Contact( "DB16000_OPC_UA_TRIGGER_ALARM".CLIENT.U02_STA3_COAXIAL.ALARMS.RESET_PC_METHOD_WORKING_BLOCKED_A )
      I_Contact( "DB16000_OPC_UA_TRIGGER_ALARM".CLIENT.U02_STA3_COAXIAL.ALARMS.READ_VARS_CONNECTION_A )
      I_Contact( "DB16000_OPC_UA_TRIGGER_ALARM".CLIENT.U02_STA3_COAXIAL.ALARMS.READ_VARS_METHOD_WORKING_BLOCKED_A )
      Not()
      Coil( #ALARM_AUX )
   END_RUNG
   RUNG wire#w1
      I_Contact( #ALARM_AUX )
      I_Contact( "DB16000_OPC_UA_TRIGGER_ALARM".CLIENT.U02_STA3_COAXIAL.ALARMS.CAMERA_FAILED_A )
      I_Contact( "DB16000_OPC_UA_TRIGGER_ALARM".CLIENT.U02_STA3_COAXIAL.ALARMS.NO_LIGHT_A )
      I_Contact( "DB16000_OPC_UA_TRIGGER_ALARM".CLIENT.U02_STA3_COAXIAL.ALARMS.CAPSULE_MISALIGNED_A )
      I_Contact( "DB16000_OPC_UA_TRIGGER_ALARM".CLIENT.U02_STA3_COAXIAL.ALARMS.JET_FAILED_ALARM )
      I_Contact( "DB16000_OPC_UA_TRIGGER_ALARM".CLIENT.U02_STA3_COAXIAL.ALARMS.NO_POWDER_A )
      I_Contact( "DB16000_OPC_UA_TRIGGER_ALARM".CLIENT.U02_STA3_COAXIAL.ALARMS.LASER_MISALIGNED_A )
      I_Contact( "DB16000_OPC_UA_TRIGGER_ALARM".CLIENT.U02_STA3_COAXIAL.ALARMS.DIRTY_CAPSULE_A )
      I_Contact( "DB16000_OPC_UA_TRIGGER_ALARM".CLIENT.U02_STA3_COAXIAL.ALARMS.DMC_STRUCTURE_A )
      Not()
      Move(in := 16015, out1 => "DB440_MACHINE_ALARM_DECODING".GLOBAL_ALARMS_MACHINE.ALARM_DECODING)
      S_Coil( "DB440_MACHINE_ALARM_DECODING".ALARMS_UNIT_02.ST3_CLADDING.IS_SEOC_ALARMS )
   END_RUNG
   // the same network as SCL:
   #ALARM_AUX := NOT ("M_ONE" AND NOT "DB16000_OPC_UA_TRIGGER_ALARM".CLIENT.U02_STA3_COAXIAL.ALARMS.CAM_START_CALIBRATION_CONNECTION_A AND NOT "DB16000_OPC_UA_TRIGGER_ALARM".CLIENT.U02_STA3_COAXIAL.ALARMS.CAM_START_CALIBRATION_METHOD_WORKING_BLOCKED_A AND NOT "DB16000_OPC_UA_TRIGGER_ALARM".CLIENT.U02_STA3_COAXIAL.ALARMS.CAM_START_ALIGNMENT_CONNECTION_A AND NOT "DB16000_OPC_UA_TRIGGER_ALARM".CLIENT.U02_STA3_COAXIAL.ALARMS.CAM_START_ALIGNMENT_METHOD_WORKING_BLOCKED_A AND NOT "DB16000_OPC_UA_TRIGGER_ALARM".CLIENT.U02_STA3_COAXIAL.ALARMS.CAM_STOP_SETUP_METHODS_CONNECTION_A AND NOT "DB16000_OPC_UA_TRIGGER_ALARM".CLIENT.U02_STA3_COAXIAL.ALARMS.CAM_STOP_SETUP_METHODS_METHOD_WORKING_BLOCKED_A AND NOT "DB16000_OPC_UA_TRIGGER_ALARM".CLIENT.U02_STA3_COAXIAL.ALARMS.CAM_START_JET_ANALISIS_CONNECTION_A AND NOT "DB16000_OPC_UA_TRIGGER_ALARM".CLIENT.U02_STA3_COAXIAL.ALARMS.CAM_START_JET_ANALISIS_METHOD_WORKING_BLOCKED_A);
   #ALARM_AUX := NOT ("M_ONE" AND NOT #ALARM_AUX AND NOT "DB16000_OPC_UA_TRIGGER_ALARM".CLIENT.U02_STA3_COAXIAL.ALARMS.CAM_START_CLADD_ANALISIS_CONNECTION_A AND NOT "DB16000_OPC_UA_TRIGGER_ALARM".CLIENT.U02_STA3_COAXIAL.ALARMS.CAM_START_CLADD_ANALISIS_METHOD_WORKING_BLOCKED_A AND NOT "DB16000_OPC_UA_TRIGGER_ALARM".CLIENT.U02_STA3_COAXIAL.ALARMS.RESET_PC_CONNECTION_A AND NOT "DB16000_OPC_UA_TRIGGER_ALARM".CLIENT.U02_STA3_COAXIAL.ALARMS.RESET_PC_METHOD_WORKING_BLOCKED_A AND NOT "DB16000_OPC_UA_TRIGGER_ALARM".CLIENT.U02_STA3_COAXIAL.ALARMS.READ_VARS_CONNECTION_A AND NOT "DB16000_OPC_UA_TRIGGER_ALARM".CLIENT.U02_STA3_COAXIAL.ALARMS.READ_VARS_METHOD_WORKING_BLOCKED_A);
   IF NOT ("M_ONE" AND NOT #ALARM_AUX AND NOT "DB16000_OPC_UA_TRIGGER_ALARM".CLIENT.U02_STA3_COAXIAL.ALARMS.CAMERA_FAILED_A AND NOT "DB16000_OPC_UA_TRIGGER_ALARM".CLIENT.U02_STA3_COAXIAL.ALARMS.NO_LIGHT_A AND NOT "DB16000_OPC_UA_TRIGGER_ALARM".CLIENT.U02_STA3_COAXIAL.ALARMS.CAPSULE_MISALIGNED_A AND NOT "DB16000_OPC_UA_TRIGGER_ALARM".CLIENT.U02_STA3_COAXIAL.ALARMS.JET_FAILED_ALARM AND NOT "DB16000_OPC_UA_TRIGGER_ALARM".CLIENT.U02_STA3_COAXIAL.ALARMS.NO_POWDER_A AND NOT "DB16000_OPC_UA_TRIGGER_ALARM".CLIENT.U02_STA3_COAXIAL.ALARMS.LASER_MISALIGNED_A AND NOT "DB16000_OPC_UA_TRIGGER_ALARM".CLIENT.U02_STA3_COAXIAL.ALARMS.DIRTY_CAPSULE_A AND NOT "DB16000_OPC_UA_TRIGGER_ALARM".CLIENT.U02_STA3_COAXIAL.ALARMS.DMC_STRUCTURE_A) THEN
       "DB440_MACHINE_ALARM_DECODING".GLOBAL_ALARMS_MACHINE.ALARM_DECODING := 16015;
       "DB440_MACHINE_ALARM_DECODING".ALARMS_UNIT_02.ST3_CLADDING.IS_SEOC_ALARMS := TRUE;
   END_IF;
END_REGION
END_FUNCTION
